PROPERTY ActualVelocity : REFERENCE TO LREAL
GET
ActualVelocity REF= lrActualVelocity;
END_GET
END_PROPERTY

PROPERTY AxisErrorID : REFERENCE TO UDINT
GET
AxisErrorID REF= iAxisErrorID;
END_GET
END_PROPERTY

PROPERTY AxisRef : AXIS_REF
GET
AxisRef := stAxisRef;
END_GET
SET
stAxisRef := AxisRef;
END_SET
END_PROPERTY

PROPERTY BufferMode : Tc2_MC2.MC_BufferMode
GET
BufferMode := eBufferMode;
END_GET
SET
eBufferMode := BufferMode;
END_SET
END_PROPERTY

PROPERTY Busy : REFERENCE TO BOOL
GET
Busy REF= bBusy;
END_GET
END_PROPERTY

PROPERTY Coupled : REFERENCE TO BOOL
GET
END_GET
END_PROPERTY

PROPERTY Deceleration : LREAL
GET
Deceleration := lrDeceleration;
END_GET
SET
lrDeceleration := Deceleration;
END_SET
END_PROPERTY

PROPERTY Direction : Tc2_MC2.MC_Direction
GET
Direction := eDirection;
END_GET
SET
eDirection := Direction;
END_SET
END_PROPERTY

PROPERTY Error : REFERENCE TO BOOL
GET
Error REF= bError;
END_GET
END_PROPERTY

PROPERTY ErrorID : REFERENCE TO UDINT
GET
ErrorID REF= iErrorID;
END_GET
END_PROPERTY

PROPERTY Halted : REFERENCE TO BOOL
GET
Halted REF= bHalted;
END_GET
END_PROPERTY

PROPERTY InPosition : REFERENCE TO BOOL
GET
InPosition REF= bInPostion;
END_GET
END_PROPERTY

PROPERTY InVelocity : REFERENCE TO BOOL
GET
InVelocity REF= bInVelocity;
END_GET
END_PROPERTY

PROPERTY IsHomed : REFERENCE TO BOOL
GET
IsHomed REF= bIsHomed;
END_GET
END_PROPERTY

PROPERTY Jerk : LREAL
GET
Jerk := lrJerk;
END_GET
SET
lrJerk := Jerk;
END_SET
END_PROPERTY

PROPERTY JogAcceleration : LREAL
GET
JogAcceleration := lrJogAcceleration;
END_GET
SET
lrJogAcceleration := JogAcceleration;
END_SET
END_PROPERTY

PROPERTY JogDeceleration : LREAL
GET
JogDeceleration := lrJogDeceleration;
END_GET
SET
lrJogDeceleration := JogDeceleration;
END_SET
END_PROPERTY

PROPERTY JogDirection : E_AxisJogDirection
GET
JogDirection := eJogDirection;
END_GET
SET
eJogDirection := JogDirection;
END_SET
END_PROPERTY

PROPERTY JogDone : REFERENCE TO BOOL
GET
JogDone REF= bJogDone;
END_GET
END_PROPERTY

PROPERTY JogJerk : LREAL
GET
JogJerk := lrJogJerk;
END_GET
SET
lrJogJerk := JogJerk;
END_SET
END_PROPERTY

PROPERTY JogMode : Tc2_MC2.E_JogMode
GET
JogMode := eJogMode;
END_GET
SET
eJogMode := JogMode;
END_SET
END_PROPERTY

PROPERTY JogPosition : LREAL
GET
JogPosition := lrJogPosition;
END_GET
SET
lrJogPosition := JogPosition;
END_SET
END_PROPERTY

PROPERTY JogVelocity : LREAL
GET
JogVelocity := lrJogVelocity;
END_GET
SET
lrJogVelocity := JogVelocity;
END_SET
END_PROPERTY

PROPERTY LagError : LREAL
GET
LagError := stAxisRef.NcToPlc.PosDiff;
END_GET
END_PROPERTY

PROPERTY Locked : REFERENCE TO BOOL
GET
Locked REF= bLocked;
END_GET
END_PROPERTY

PROPERTY MoveActive : REFERENCE TO BOOL
GET
MoveActive REF= bMoveActive;
END_GET
END_PROPERTY

METHOD MR_Abort : BOOL
IF eAxisState >= AXIS_INITIALIZING THEN
	bAbort := TRUE;
	eAxisState := AXIS_ABORTING;
	fbMachineLogger.MR_AddLogs(CONCAT(sName,' : abort requested'));
	
ELSIF eAxisState = AXIS_UNINITIALIZED THEN
	bAbort 		:= FALSE;
	MR_Abort	:= TRUE;
	fbMachineLogger.MR_AddLogs(CONCAT(sName,' : abort done'));
	
END_IF
END_METHOD

METHOD MR_Couple : BOOL
VAR_INPUT
END_VAR
;
END_METHOD

METHOD MR_Decouple : BOOL
VAR_INPUT
END_VAR
;
END_METHOD

METHOD MR_FirstCycle
VAR_INPUT
	sName 				: STRING; 	(* Axis object name *)
	sMeasurementUnits	: STRING;	(* Measurement units used by axis *)
	bModulo				: BOOL;		(* Axis is periodic *)
END_VAR
THIS^.sName := sName;
THIS^.sUnit := sMeasurementUnits;
THIS^.bModulo := bModulo;
END_METHOD

METHOD MR_Halt : BOOL
IF eAxisState >= AXIS_IDLE AND eAxisState <> AXIS_HALT_DONE THEN
	IF NOT bHaltLog THEN 
		fbMachineLogger.MR_AddLogs(CONCAT(sName,' : halt requested'));
		bHaltLog := TRUE;
	END_IF
	
	bHalt := TRUE;
	eAxisState := AXIS_HALT;
	
ELSIF eAxisState = AXIS_HALT_DONE THEN
	bInPostion 	:= FALSE;
	bInVelocity := FALSE;
	bMoveActive := FALSE;
	bStopped 	:= FALSE;
	bHalted 	:= TRUE;
	bJogDone 	:= FALSE;
	
	bHalt		:= FALSE;
	MR_Halt 	:= TRUE;

	bHaltLog 	:= FALSE;
	fbMachineLogger.MR_AddLogs(CONCAT(sName,' : halt done'));
	
END_IF
END_METHOD

METHOD MR_Home : BOOL
VAR_INPUT
	lrHomePosition : LREAL;
END_VAR
IF eAxisState = AXIS_IDLE THEN
	THIS^.lrHomePosition := lrHomePosition;
	bIsHomed := FALSE;
	
	bHome := TRUE;
	eAxisState := AXIS_HOME;
	fbMachineLogger.MR_AddLogs(CONCAT(sName,' : home position requested'));
	
ELSIF eAxisState = AXIS_HOME_DONE THEN
	bIsHomed := TRUE;
	
	bHome := FALSE;
	MR_Home := TRUE;
	fbMachineLogger.MR_AddLogs(CONCAT(sName,' : home position done'));	
	
END_IF
END_METHOD

METHOD MR_Init : BOOL
IF eAxisState = AXIS_UNINITIALIZED THEN
	bInit := TRUE;
	fbMachineLogger.MR_AddLogs(CONCAT(sName,' : initialization requested'));
	
ELSIF eAxisState = AXIS_INITIALIZING AND eAxisStateInit = AXIS_INIT_DONE THEN
	//bPowerOn 	:= TRUE;
	bInPostion 	:= FALSE;
	bInVelocity := FALSE;
	bMoveActive := FALSE;
	bStopped 	:= FALSE;
	bHalted 	:= FALSE;
	bJogDone 	:= FALSE;

	bInit 		:= FALSE;
	MR_Init 	:= TRUE;
	
	fbMachineLogger.MR_AddLogs(CONCAT(sName,' : initialization done'));

END_IF
END_METHOD

METHOD MR_Jog : BOOL
VAR_INPUT
	bJogActive	  : BOOL;
END_VAR
THIS^.bJogActive := bJogActive;

IF eAxisState = AXIS_IDLE THEN
	bJog := TRUE;
	bInPostion 	:= FALSE;
	bInVelocity	:= FALSE;
	bMoveActive	:= TRUE;
	bStopped	:= FALSE;
	bHalted 	:= FALSE;
	bJogDone 	:= FALSE;
	
	eAxisState := AXIS_MOVE_JOG;
	fbMachineLogger.MR_AddLogs(CONCAT(sName,' : move jog requested'));	
	
ELSIF eAxisState = AXIS_MOVE_JOG_DONE THEN
	IF eJogMode = E_JogMode.MC_JOGMODE_INCHING OR eJogMode = E_JogMode.MC_JOGMODE_INCHING_MODULO THEN
		bInPostion 	:= TRUE;
	END_IF
	
	bInVelocity := FALSE;
	bMoveActive := FALSE;
	bStopped 	:= FALSE;
	bHalted 	:= FALSE;
	bJogDone 	:= TRUE;	

	bJog 		:= FALSE;
	MR_Jog 		:= TRUE;
	
	fbMachineLogger.MR_AddLogs(CONCAT(sName,' : move jog done'));		
	
END_IF
END_METHOD

METHOD MR_MoveAbsolute : BOOL
VAR_INPUT
	lrAbsolutePosition : LREAL;
END_VAR
IF eAxisState = AXIS_IDLE AND THIS^.lrActualPosition <> lrAbsolutePosition THEN
	THIS^.lrAbsolutePosition := lrAbsolutePosition;
	bMoveAbsolute := TRUE;
	bInPostion 	:= FALSE;
	bInVelocity := FALSE;
	bMoveActive := TRUE;
	bStopped 	:= FALSE;
	bHalted 	:= FALSE;
	bJogDone 	:= FALSE;
	
	eAxisState := AXIS_MOVE_ABSOLUTE;
	fbMachineLogger.MR_AddLogs(CONCAT(sName,' : move absolute requested'));		
	
ELSIF eAxisState = AXIS_MOVE_ABSOLUTE_DONE THEN
	bInPostion 		:= TRUE;
	bInVelocity		:= FALSE;
	bMoveActive 	:= FALSE;
	bStopped 		:= FALSE;
	bHalted			:= FALSE;
	bJogDone 		:= FALSE;
	
	bMoveAbsolute 	:= FALSE;
	MR_MoveAbsolute := TRUE;
	fbMachineLogger.MR_AddLogs(CONCAT(sName,' : move absolute done'));		
	
END_IF
END_METHOD

METHOD MR_MoveAdditive : BOOL
VAR_INPUT
	lrRelativeDistance : LREAL;
END_VAR
THIS^.lrRelativeDistance := lrRelativeDistance;
IF eAxisState = AXIS_IDLE AND THIS^.lrRelativeDistance <> 0.0 THEN
	bMoveAdditive := TRUE;
	bInPostion 	:= FALSE;
	bInVelocity := FALSE;
	bStopped 	:= FALSE;
	bHalted 	:= FALSE;
	bJogDone 	:= FALSE;
	
	bMoveActive := TRUE;
	eAxisState := AXIS_MOVE_ADDITIVE;
	fbMachineLogger.MR_AddLogs(CONCAT(sName,' : move additive requested'));		
	
ELSIF eAxisState = AXIS_MOVE_ADDITIVE_DONE THEN
	bInPostion 		:= TRUE;
	bInVelocity 	:= FALSE;
	bStopped 		:= FALSE;
	bHalted 		:= FALSE;
	bJogDone 		:= FALSE;
	
	bMoveAdditive 	:= FALSE;
	MR_MoveAdditive := TRUE;
	fbMachineLogger.MR_AddLogs(CONCAT(sName,' : move additive done'));		
	
END_IF
END_METHOD

METHOD MR_MoveRelative : BOOL
VAR_INPUT
	lrRelativeDistance : LREAL;
END_VAR
THIS^.lrRelativeDistance := lrRelativeDistance;
IF eAxisState = AXIS_IDLE AND THIS^.lrRelativeDistance <> 0.0 THEN
	bMoveRelative := TRUE;
	bInPostion 	:= FALSE;
	bInVelocity := FALSE;
	bMoveActive := TRUE;
	bStopped 	:= FALSE;
	bHalted 	:= FALSE;
	bJogDone 	:= FALSE;
	
	eAxisState := AXIS_MOVE_RELATIVE;
	fbMachineLogger.MR_AddLogs(CONCAT(sName,' : move relative requested'));			
	
ELSIF eAxisState = AXIS_MOVE_RELATIVE_DONE THEN
	bMoveRelative 	:= FALSE;
	MR_MoveRelative := TRUE;
	
	bInPostion 		:= TRUE;
	bInVelocity 	:= FALSE;
	bMoveActive 	:= FALSE;
	bStopped 		:= FALSE;
	bHalted 		:= FALSE;
	bJogDone 		:= FALSE;
	
	fbMachineLogger.MR_AddLogs(CONCAT(sName,' : move relative done'));		
	
END_IF
END_METHOD

METHOD MR_MoveVelocity : BOOL
IF eAxisState = AXIS_IDLE THEN
	bMoveVelocity 	:= TRUE;
	bInPostion 		:= FALSE;
	bInVelocity 	:= FALSE;
	bMoveActive 	:= TRUE;
	bStopped 		:= FALSE;
	bHalted 		:= FALSE;
	bJogDone 		:= FALSE;	
	
	eAxisState 		:= AXIS_MOVE_VELOCITY;
	fbMachineLogger.MR_AddLogs(CONCAT(sName,' : move velocity requested'));			
	
ELSIF eAxisState = AXIS_MOVE_VELOCITY_DONE THEN
	bMoveVelocity 	:= FALSE;
	MR_MoveVelocity := TRUE;
	
	bInPostion 		:= FALSE;
	bInVelocity 	:= TRUE;
	bMoveActive 	:= TRUE;
	bStopped 		:= FALSE;
	bHalted 		:= FALSE;
	bJogDone 		:= FALSE;
	
	fbMachineLogger.MR_AddLogs(CONCAT(sName,' : move velocity done'));		
	
END_IF
END_METHOD

METHOD MR_Reset : BOOL
IF eAxisState <> AXIS_RESET AND eAxisState <> AXIS_RESET_DONE AND bError THEN
	bReset := TRUE;
	eAxisStateBeforeReset := eAxisState;
	eAxisState := AXIS_RESET;
	fbMachineLogger.MR_AddLogs(CONCAT(sName,' : reset requested'));			
	
ELSIF eAxisState = AXIS_RESET_DONE THEN
	bError := FALSE;
	iErrorID := 0;
	
	bReset := FALSE;
	MR_Reset := TRUE;
	
	fbMachineLogger.MR_AddLogs(CONCAT(sName,' : reset done'));		
		
END_IF
END_METHOD

METHOD MR_Stop : BOOL
IF eAxisState >= AXIS_IDLE AND eAxisState <> AXIS_STOP_DONE THEN
	IF NOT bStopLog THEN 
		fbMachineLogger.MR_AddLogs(CONCAT(sName,' : stop requested'));
		bStopLog := TRUE;	
	END_IF
	
	bStop := TRUE;
	eAxisState := AXIS_STOP;
	
ELSIF eAxisState = AXIS_STOP_DONE THEN
	bStop 		:= FALSE;
	MR_Stop 	:= TRUE;
	
	bInPostion 	:= FALSE;
	bInVelocity := FALSE;
	bMoveActive := FALSE;
	bStopped 	:= TRUE;
	bHalted 	:= FALSE;
	bJogDone 	:= FALSE;
	bLocked		:= TRUE;
	
	bStopLog 	:= FALSE;
	fbMachineLogger.MR_AddLogs(CONCAT(sName,' : stop done'));			
END_IF
END_METHOD

METHOD MR_Unlock : BOOL
VAR_INPUT
END_VAR
IF eAxisState = AXIS_IDLE THEN
	bUnlock := TRUE;
	MR_Unlock := FALSE;
	eAxisState := AXIS_UNLOCK;
	fbMachineLogger.MR_AddLogs(CONCAT(sName,' : unlock after stop requested'));
	
ELSIF eAxisState = AXIS_UNLOCK_DONE THEN
	bUnlock := FALSE;
	MR_Unlock := TRUE;
	bLocked := FALSE;
	fbMachineLogger.MR_AddLogs(CONCAT(sName,' : unlock after stop done'));
	
END_IF
END_METHOD

METHOD PROTECTED MS_Aborting
VAR_INPUT
END_VAR
(* Reset MC_Halt *)
fbMcHalt( Axis := stAxisRef, Execute := FALSE);

(* Reset MC_Stop *)
fbMcStop( Axis := stAxisRef, Execute := FALSE);

(* Reset MC_MoveVelocity *)
fbMcMoveVelocity( Axis := stAxisRef, Execute := FALSE);

(* Reset MC_MoveAbsolute *)
fbMcMoveAbsolute( Axis := stAxisRef, Execute := FALSE);

(* Reset MC_MoveAdditive *)
fbMcMoveAdditive( Axis := stAxisRef, Execute := FALSE);

(* Reset MC_MoveRelative *)
fbMcMoveRelative( Axis := stAxisRef, Execute := FALSE);

(* Reset MC_Jog *)
fbMcJog( Axis := stAxisRef, JogForward := FALSE ,JogBackwards := FALSE);

(* Reset MC_Reset *)
fbMcReset( Axis := stAxisRef, Execute := FALSE);

(* Reset MC_Power *)
fbMcPower(	Enable 			:= FALSE,
			Enable_Positive := FALSE,
			Enable_Negative := FALSE,
			Override 		:= lrOverride,
			Axis 			:= stAxisRef);
					
IF fbReadAxisStatus.Disabled AND NOT fbMcStop.Busy THEN
	bInPostion	:= FALSE;
	bInVelocity := FALSE;
	bMoveActive := FALSE;
	bStopped 	:= FALSE;
	bHalted 	:= FALSE;
	bJogDone	:= FALSE;
	bIsHomed 	:= FALSE;
	bLocked		:= FALSE;
	eAxisState	:= AXIS_UNINITIALIZED;	
	
END_IF
END_METHOD

METHOD PROTECTED MS_Couple : BOOL
VAR_INPUT
END_VAR
(*
IF NOT fbMcGearIn.Error THEN
	fbMcGearIn( Master				:=,
				Slave 				:= ,
				Execute 			:= TRUE,
				RatioNumerator		:=,
				RatioDenominator 	:=,
				Acceleration 		:= ,
				Deceleration 		:= ,
				Jerk 				:=,
				BufferMode 			:=,
				Options				:=);
				
	IF fbMcGearIn.InGear THEN
		eAxisState := AXIS_COUPLE_DONE;
	END_IF
ELSE
	bError := TRUE;
	iErrorID := fbMcGearIn.ErrorID;
	fbMcGearIn( Master := , Slave := , Execute := FALSE);
	fbAlarmCoupling.ipArguments.Clear().AddUDInt(iErrorID);
	fbAlarmCoupling.Raise(0);
END_IF
*)
END_METHOD

METHOD MS_CoupleDone : BOOL
VAR_INPUT
END_VAR
END_METHOD

METHOD MS_Decouple : BOOL
VAR_INPUT
END_VAR
(*
IF NOT fbMcGearOut.Error THEN			
	fbMcGearOut( 	Slave 	:=,
					Execute := TRUE,
					Options := );	
				
	IF fbMcGearOut.Done THEN
		eAxisState := AXIS_DECOUPLE_DONE;
	END_IF
ELSE
	bError := TRUE;
	iErrorID := fbMcGearOut.ErrorID;
	fbMcGearOut( Slave := , Execute := FALSE);
	fbAlarmDecoupling.ipArguments.Clear().AddUDInt(iErrorID);
	fbAlarmDecoupling.Raise(0);
END_IF
*)
END_METHOD

METHOD MS_DecoupleDone : BOOL
VAR_INPUT
END_VAR
END_METHOD

METHOD MS_Extension : BOOL
VAR_INPUT
END_VAR
END_METHOD

METHOD PROTECTED MS_Halt
VAR_INPUT
END_VAR
(* Reset MC_MoveVelocity *)
fbMcMoveVelocity( Axis := stAxisRef, Execute := FALSE);

(* Reset MC_MoveAbsolute *)					
fbMcMoveAbsolute( Axis := stAxisRef, Execute := FALSE);

(* Reset MC_MoveAdditive *)					
fbMcMoveAdditive( Axis := stAxisRef ,Execute := FALSE);

(* Reset MC_MoveRelative *)					
fbMcMoveRelative( Axis := stAxisRef, Execute := FALSE);

(* Reset MC_Jog *)
fbMcJog( Axis := stAxisRef, JogForward := FALSE, JogBackwards := FALSE);

fbMcHalt(	Axis			:= stAxisRef,
			Execute 		:= TRUE,
			Deceleration 	:= lrDeceleration,
			Jerk 			:= lrJerk,
			BufferMode 		:= MC_Aborting);

IF fbMcHalt.Error THEN
	bError := TRUE;
	iErrorID := fbMcHalt.ErrorID;
	fbMcHalt(Axis := stAxisRef, Execute := FALSE);
	fbAlarmHalt.ipArguments.Clear().AddUDInt(iErrorID);
	fbAlarmHalt.Raise(0);

ELSIF fbMcHalt.Done THEN
	eAxisState := AXIS_HALT_DONE;
END_IF
END_METHOD

METHOD PROTECTED MS_HaltDone
VAR_INPUT
END_VAR
fbMcHalt( Axis := stAxisRef, Execute := FALSE);

IF NOT bHalt AND NOT fbMcHalt.Busy THEN
	eAxisState := AXIS_IDLE;
END_IF
END_METHOD

METHOD PROTECTED ABSTRACT MS_Home
VAR_INPUT
END_VAR
END_METHOD

METHOD PROTECTED ABSTRACT MS_HomeDone
VAR_INPUT
END_VAR
END_METHOD

METHOD PROTECTED MS_Idle
VAR_INPUT
END_VAR
;
END_METHOD

METHOD PROTECTED MS_Initializing
VAR_INPUT
END_VAR
CASE eAxisStateInit OF
	AXIS_INIT_RESET:
		fbMcReset(	Execute := TRUE, Axis := stAxisRef);
		
		IF fbMcReset.Error THEN
			bError := fbMcReset.Error;
			iErrorID := fbMcReset.ErrorID;
			fbMcReset(Axis := stAxisRef, Execute := FALSE);
			fbAlarmInitReset.ipArguments.Clear().AddUDInt(iErrorID);
			fbAlarmInitReset.Raise(0);
			
		ELSIF fbMcReset.Done THEN
			fbMcReset(Axis := stAxisRef, Execute := FALSE);
			eAxisStateInit := AXIS_INIT_POWER_ON;
			
		END_IF
		
	AXIS_INIT_POWER_ON:
		fbMcPower(	Enable 			:= TRUE,
					Enable_Positive := TRUE,
					Enable_Negative := TRUE,
					Override 		:= lrOverride,
					Axis 			:= stAxisRef);
			
		IF fbMcPower.Error THEN
			bError := fbMcPower.Error;
			iErrorID := fbMcPower.ErrorID;
			fbAlarmInitPowerOn.ipArguments.Clear().AddUDInt(iErrorID);
			fbAlarmInitPowerOn.Raise(0);			
			
		ELSIF fbMcPower.Status THEN
			eAxisStateInit := AXIS_INIT_DONE;	
				
		END_IF
	
	AXIS_INIT_DONE:
		IF NOT bInit THEN
			eAxisState := AXIS_READY_INITIALIZED;
		END_IF
END_CASE
END_METHOD

METHOD PROTECTED MS_MoveAbsolute
VAR_INPUT
END_VAR
fbMcMoveAbsolute(	Axis			:= stAxisRef,
					Execute 		:= TRUE,
					Position 		:= lrAbsolutePosition,
					Velocity 		:= lrVelocity,
					Acceleration 	:= lrAcceleration,
					Deceleration 	:= lrDeceleration,
					Jerk 			:= lrJerk,
					BufferMode 		:= eBufferMode);

IF fbMcMoveAbsolute.Error THEN
	bError := TRUE;
	bMoveActive := FALSE;
	iErrorID := fbMcMoveAbsolute.ErrorID;
	fbMcMoveAbsolute( Axis := stAxisRef, Execute := FALSE);
	fbAlarmMoveAbsolute.ipArguments.Clear().AddUDInt(iErrorID);
	fbAlarmMoveAbsolute.Raise(0);

ELSIF fbMcMoveAbsolute.Done THEN
	eAxisState := AXIS_MOVE_ABSOLUTE_DONE;
END_IF
END_METHOD

METHOD PROTECTED MS_MoveAbsoluteDone
VAR_INPUT
END_VAR
fbMcMoveAbsolute( Axis := stAxisRef, Execute := FALSE);

IF NOT bMoveAbsolute AND NOT fbMcMoveAbsolute.Busy THEN
	eAxisState := AXIS_IDLE;
END_IF
END_METHOD

METHOD PROTECTED MS_MoveAdditive
VAR_INPUT
END_VAR
fbMcMoveAdditive(	Axis			:= stAxisRef,
					Execute 		:= TRUE,
					Distance 		:= lrRelativeDistance,
					Velocity		:= lrVelocity,
					Acceleration	:= lrAcceleration,
					Deceleration	:= lrDeceleration,
					Jerk			:= lrJerk,
					BufferMode 		:= eBufferMode);

IF fbMcMoveAdditive.Error THEN
	bError := TRUE;
	bMoveActive := FALSE;
	iErrorID := fbMcMoveAdditive.ErrorID;
	fbMcMoveAdditive( Axis := stAxisRef, Execute := FALSE);
	fbAlarmMoveAdditive.ipArguments.Clear().AddUDInt(iErrorID);
	fbAlarmMoveAdditive.Raise(0);
		
ELSIF fbMcMoveAdditive.Done THEN
	eAxisState := AXIS_MOVE_ADDITIVE_DONE;
END_IF
END_METHOD

METHOD PROTECTED MS_MoveAdditiveDone
VAR_INPUT
END_VAR
fbMcMoveAdditive( Axis := stAxisRef, Execute := FALSE);

IF NOT bMoveAdditive AND NOT fbMcMoveAdditive.Busy THEN
	eAxisState := AXIS_IDLE;
END_IF
END_METHOD

METHOD PROTECTED MS_MoveJog
VAR_INPUT
END_VAR
VAR
	bJogForward: BOOL;
	bJogBackward: BOOL;
END_VAR
IF eJogDirection = AXIS_JOG_DIR_POSITIVE THEN
	bJogForward := TRUE;
	bJogBackward:= FALSE;
	
ELSIF eJogDirection = AXIS_JOG_DIR_NEGATIVE THEN
	bJogForward := FALSE;
	bJogBackward:= TRUE;
		
END_IF

fbMcJog( 	Axis 			:= stAxisRef,
			JogForward		:= bJogForward,
			JogBackwards	:= bJogBackward,
			Mode 			:= eJogMode,
			Position 		:= lrJogPosition,
			Velocity 		:= lrJogVelocity,
			Acceleration 	:= lrJogAcceleration,
			Deceleration 	:= lrJogDeceleration,
			Jerk 			:= lrJogJerk);

IF fbMcJog.Error THEN
	bError := TRUE;
	bMoveActive := FALSE;
	iErrorID := fbMcJog.ErrorID;
	fbMcJog( Axis := stAxisRef, JogForward := FALSE, JogBackwards := FALSE);
	fbAlarmMoveJog.ipArguments.Clear().AddUDInt(iErrorID);
	fbAlarmMoveJog.Raise(0);
	
ELSIF fbMcJog.Mode >= MC_JOGMODE_INCHING AND fbMcJog.Done THEN
	eAxisState := AXIS_MOVE_JOG_DONE;
		
ELSIF fbMcJog.Mode < MC_JOGMODE_INCHING AND NOT bJogActive THEN
	eAxisState := AXIS_MOVE_JOG_DONE;
		
END_IF
END_METHOD

METHOD PROTECTED MS_MoveJogDone
VAR_INPUT
END_VAR
fbMcJog( Axis := stAxisRef, JogForward := FALSE, JogBackwards := FALSE);

IF NOT bJog AND NOT fbMcJog.Busy THEN
	eAxisState := AXIS_IDLE;
END_IF
END_METHOD

METHOD PROTECTED MS_MoveRelative
VAR_INPUT
END_VAR
fbMcMoveRelative(	Axis 			:= stAxisRef,
					Execute 		:= TRUE,
					Distance 		:= lrRelativeDistance,
					Velocity 		:= lrVelocity,
					Acceleration 	:= lrAcceleration,
					Deceleration 	:= lrDeceleration,
					Jerk 			:= lrJerk,
					BufferMode 		:= eBufferMode);
				
IF fbMcMoveRelative.Error THEN
	bError := TRUE;
	iErrorID := fbMcMoveRelative.ErrorID;
	fbMcMoveRelative( Axis := stAxisRef, Execute := FALSE);
	fbAlarmMoveRelative.ipArguments.Clear().AddUDInt(iErrorID);
	fbAlarmMoveRelative.Raise(0);
	
ELSIF fbMcMoveRelative.Done THEN
	eAxisState := AXIS_MOVE_RELATIVE_DONE;
END_IF
END_METHOD

METHOD PROTECTED MS_MoveRelativeDone
VAR_INPUT
END_VAR
fbMcMoveRelative( Axis := stAxisRef, Execute := FALSE);

IF NOT bMoveRelative AND NOT fbMcMoveRelative.Busy THEN
	bInPostion := TRUE;
	bInVelocity := FALSE;
	bMoveActive := FALSE;
	bStopped := FALSE;
	bHalted := FALSE;
	bJogDone := FALSE;
	eAxisState := AXIS_IDLE;
END_IF
END_METHOD

METHOD PROTECTED MS_MoveVelocity
VAR_INPUT
END_VAR
fbMcMoveVelocity(	Axis 			:= stAxisRef,
					Execute 		:= TRUE,
					Velocity 		:= lrVelocity,
					Acceleration 	:= lrAcceleration,
					Deceleration 	:= lrDeceleration,
					Jerk 			:= lrJerk,
					Direction 		:= eDirection,
					BufferMode 		:= eBufferMode);

IF fbMcMoveVelocity.Error THEN
	bError := TRUE;
	iErrorID := fbMcMoveVelocity.ErrorID;
	fbMcMoveVelocity( Axis := stAxisRef, Execute := FALSE);
	fbAlarmMoveVelocity.ipArguments.Clear().AddUDInt(iErrorID);
	fbAlarmMoveVelocity.Raise(0);
	
ELSIF fbMcMoveVelocity.InVelocity THEN
	eAxisState := AXIS_MOVE_VELOCITY_DONE;
END_IF
END_METHOD

METHOD PROTECTED MS_MoveVelocityDone
VAR_INPUT
END_VAR
fbMcMoveVelocity( Axis := stAxisRef, Execute := FALSE);

IF NOT bMoveVelocity AND NOT fbMcMoveVelocity.Busy THEN
	eAxisState := AXIS_IDLE;
END_IF
END_METHOD

METHOD PROTECTED MS_ReadyInitialized
VAR_INPUT
END_VAR
eAxisState := AXIS_IDLE;
END_METHOD

METHOD PROTECTED MS_Reset
VAR_INPUT
END_VAR
(* Reset MC_Halt *)
fbMcHalt( Axis := stAxisRef, Execute := FALSE);

(* Reset MC_Stop *)
fbMcStop( Axis := stAxisRef, Execute := FALSE);

(* Reset MC_MoveVelocity *)
fbMcMoveVelocity( Axis := stAxisRef, Execute := FALSE);

(* Reset MC_MoveAbsolute *)
fbMcMoveAbsolute( Axis := stAxisRef, Execute := FALSE);

(* Reset MC_MoveAdditive *)
fbMcMoveAdditive( Axis := stAxisRef, Execute := FALSE);

(* Reset MC_MoveRelative *)
fbMcMoveRelative( Axis := stAxisRef, Execute := FALSE);

(* Reset MC_Jog *)
fbMcJog( Axis := stAxisRef, JogForward := FALSE ,JogBackwards := FALSE);

(* Reset MC_GearIn *)
;

(* Reset MC_GearOut *)
;

(* Reset internal commands *)
bAbort			:= FALSE;
bHalt 			:= FALSE;
bHome			:= FALSE;
bJog			:= FALSE;
bMoveAbsolute	:= FALSE;
bMoveAdditive	:= FALSE;
bMoveRelative	:= FALSE;
bMoveVelocity	:= FALSE;
bStop			:= FALSE;

fbMcReset( Axis := stAxisRef, Execute := TRUE);

IF fbMcReset.Error THEN
	bError := TRUE;
	iErrorID := fbMcReset.ErrorID;
	fbMcReset( Axis := stAxisRef, Execute := FALSE);
	fbAlarmInitReset.ipArguments.Clear().AddUDInt(iErrorID);
	fbAlarmInitReset.Raise(0);
	
ELSIF fbMcReset.Done THEN
	fbMcReset(Axis := stAxisRef, Execute := FALSE);
	
	(* Confirming and resetting alarms *)
	fbAlarmHalt.Confirm(nTimeStamp := 0);
	fbAlarmInitReset.Confirm(nTimeStamp := 0);
	fbAlarmInitPowerOn.Confirm(nTimeStamp := 0);
	fbAlarmMoveAbsolute.Confirm(nTimeStamp := 0);
	fbAlarmMoveAdditive.Confirm(nTimeStamp := 0);
	fbAlarmMoveJog.Confirm(nTimeStamp := 0);
	fbAlarmMoveRelative.Confirm(nTimeStamp := 0);
	fbAlarmMoveVelocity.Confirm(nTimeStamp := 0);
	fbAlarmStop.Confirm(nTimeStamp := 0);
	fbAlarmHome.Confirm(nTimeStamp := 0);
	fbAlarmHaltCA.Confirm(nTimeStamp := 0);
	fbAlarmMoveAbsoluteCA.Confirm(nTimeStamp := 0);
	fbAlarmMoveRelativeCA.Confirm(nTimeStamp := 0);
	fbAlarmCoupling.Confirm(nTimeStamp := 0);
	fbAlarmDecoupling.Confirm(nTimeStamp := 0);

	fbAlarmHalt.Clear(nTimeStamp := 0, bResetConfirmation := bResetConfirmation); 
	fbAlarmInitReset.Clear(nTimeStamp := 0, bResetConfirmation := bResetConfirmation); 
	fbAlarmInitPowerOn.Clear(nTimeStamp := 0, bResetConfirmation := bResetConfirmation); 
	fbAlarmMoveAbsolute.Clear(nTimeStamp := 0, bResetConfirmation := bResetConfirmation); 
	fbAlarmMoveAdditive.Clear(nTimeStamp := 0, bResetConfirmation := bResetConfirmation); 
	fbAlarmMoveJog.Clear(nTimeStamp := 0, bResetConfirmation := bResetConfirmation); 
	fbAlarmMoveRelative.Clear(nTimeStamp := 0, bResetConfirmation := bResetConfirmation); 
	fbAlarmMoveVelocity.Clear( nTimeStamp := 0, bResetConfirmation := bResetConfirmation); 
	fbAlarmStop.Clear(nTimeStamp := 0, bResetConfirmation := bResetConfirmation); 
	fbAlarmHome.Clear(nTimeStamp := 0, bResetConfirmation := bResetConfirmation); 
	fbAlarmHaltCA.Clear(nTimeStamp := 0, bResetConfirmation := bResetConfirmation); 
	fbAlarmMoveAbsoluteCA.Clear(nTimeStamp := 0, bResetConfirmation := bResetConfirmation); 
	fbAlarmMoveRelativeCA.Clear(nTimeStamp := 0, bResetConfirmation := bResetConfirmation); 
	fbAlarmCoupling.Clear(nTimeStamp := 0, bResetConfirmation := bResetConfirmation); 
	fbAlarmDecoupling.Clear(nTimeStamp := 0, bResetConfirmation := bResetConfirmation); 

	IF NOT fbMcHalt.Busy AND NOT fbMcStop.Busy AND NOT fbMcMoveVelocity.Busy AND
		NOT fbMcMoveAbsolute.Busy AND NOT fbMcMoveAdditive.Busy AND NOT fbMcMoveRelative.Busy AND NOT fbMcReset.Busy THEN
		eAxisState := AXIS_RESET_DONE;
	END_IF
END_IF
END_METHOD

METHOD PROTECTED MS_ResetDone
VAR_INPUT
END_VAR
IF NOT bReset THEN
	IF eAxisStateBeforeReset >= E_AxisState.AXIS_IDLE THEN
		eAxisState := AXIS_IDLE;
	ELSE
		eAxisState := AXIS_UNINITIALIZED;	
	END_IF
END_IF
END_METHOD

METHOD PROTECTED MS_Stop
VAR_INPUT
END_VAR
(* Reset MC_MoveVelocity *)
fbMcMoveVelocity( Axis := stAxisRef, Execute := FALSE);

(* Reset MC_MoveAbsolute *)					
fbMcMoveAbsolute( Axis := stAxisRef, Execute := FALSE);

(* Reset MC_MoveAdditive *)					
fbMcMoveAdditive( Axis := stAxisRef ,Execute := FALSE);

(* Reset MC_MoveRelative *)					
fbMcMoveRelative( Axis := stAxisRef, Execute := FALSE);

(* Reset MC_Jog *)
fbMcJog( Axis := stAxisRef, JogForward := FALSE, JogBackwards := FALSE);

fbMcStop(	Execute 		:= TRUE,
			Axis 			:= stAxisRef,
			Deceleration	:= lrStopDeceleration,
			Jerk 			:= lrStopJerk);

IF fbMcStop.Error THEN
	bError := TRUE;
	iErrorID := fbMcStop.ErrorID;
	fbMcStop( Axis := stAxisRef, Execute := FALSE);
	fbAlarmStop.ipArguments.Clear().AddUDInt(iErrorID);
	fbAlarmStop.Raise(0);
	
ELSIF fbMcStop.Done THEN
	eAxisState := AXIS_STOP_DONE;
END_IF
END_METHOD

METHOD PROTECTED MS_StopDone
VAR_INPUT
END_VAR
fbMcStop( Axis := stAxisRef, Execute := FALSE);

IF NOT bStop THEN
	eAxisState := AXIS_IDLE;	
END_IF
END_METHOD

METHOD PROTECTED MS_Uninitalized
VAR_INPUT
END_VAR
(* Reset all commands *)
bAbort				:= FALSE;
bHalt 				:= FALSE;
bHome				:= FALSE;
bJog				:= FALSE;
bMoveAbsolute		:= FALSE;
bMoveAdditive		:= FALSE;
bMoveRelative		:= FALSE;
bMoveVelocity		:= FALSE;
bReset				:= FALSE;
bStop				:= FALSE;

(* Reset status flags *)
bError				:= FALSE;
bInPostion			:= FALSE;
bInVelocity			:= FALSE;
bIsHomed			:= FALSE;
bMoveActive			:= FALSE;
bPowerOn			:= FALSE;
bStopped			:= FALSE;
bJogDone			:= FALSE;
bLocked				:= FALSE;
lrActualPosition 	:= 0.0;
lrActualVelocity 	:= 0.0;
iErrorID			:= 0;

IF bInit THEN
	eAxisState := AXIS_INITIALIZING;
	eAxisStateInit := AXIS_INIT_RESET;	
END_IF
END_METHOD

METHOD MS_Unlock
VAR_INPUT
END_VAR
fbMcStop( Axis := stAxisRef, Execute := FALSE);

IF NOT fbMcStop.Busy THEN
	eAxisState := AXIS_UNLOCK_DONE;
END_IF
END_METHOD

METHOD MS_UnlockDone
VAR_INPUT
END_VAR
IF NOT bUnlock THEN
	eAxisState := AXIS_IDLE;
END_IF
END_METHOD

PROPERTY Name : STRING
GET
Name := sName;
END_GET
SET
sName := Name;
END_SET
END_PROPERTY

PROPERTY Options : Tc2_MC2.ST_MoveOptions
GET
Options := stOptions;
END_GET
SET
stOptions := Options;
END_SET
END_PROPERTY

PROPERTY Override : LREAL
GET
Override := lrOverride;
END_GET
SET
IF Override >= 0.0 AND Override <= 200.0 THEN
	lrOverride := Override;
	fbMcPower( Axis := stAxisRef, Override := lrOverride);
END_IF
END_SET
END_PROPERTY

PROPERTY PowerOn : REFERENCE TO BOOL
GET
PowerOn REF= bPowerOn;
END_GET
END_PROPERTY

PROPERTY SetpointPosition : LREAL
GET
SetpointPosition := stAxisRef.NcToPlc.SetPos;
END_GET
END_PROPERTY

PROPERTY SetpointVelocity : LREAL
GET
SetpointVelocity := stAxisRef.NcToPlc.SetVelo;
END_GET
END_PROPERTY

PROPERTY State : REFERENCE TO E_AxisState
GET
State REF= eAxisState;
END_GET
END_PROPERTY

METHOD PROTECTED StateMachine
VAR_INPUT
END_VAR

VAR

END_VAR
CASE eAxisState OF
	AXIS_UNINITIALIZED:
		MS_Uninitalized();
		
	AXIS_INITIALIZING:
		MS_Initializing();
		
	AXIS_READY_INITIALIZED:
		MS_ReadyInitialized();
		
	AXIS_IDLE:
		MS_Idle();
	
	AXIS_HOME:
		MS_Home();
		
	E_AxisState.AXIS_HOME_DONE:
		MS_HomeDone();
		
	AXIS_MOVE_VELOCITY:
		MS_MoveVelocity();
	
	AXIS_MOVE_VELOCITY_DONE:
		MS_MoveVelocityDone();
	
	AXIS_MOVE_ABSOLUTE:
		MS_MoveAbsolute();
	
	AXIS_MOVE_ABSOLUTE_DONE:
		MS_MoveAbsoluteDone();
	
	AXIS_MOVE_ADDITIVE:
		MS_MoveAdditive();
	
	AXIS_MOVE_ADDITIVE_DONE:
		MS_MoveAdditiveDone();
		
	AXIS_MOVE_RELATIVE:
		MS_MoveRelative();
		
	AXIS_MOVE_RELATIVE_DONE:
		MS_MoveRelativeDone();
	
	AXIS_MOVE_JOG:
		MS_MoveJog();
	
	AXIS_MOVE_JOG_DONE:
		MS_MoveJogDone();
	
	AXIS_STOP:
		MS_Stop();
	
	AXIS_STOP_DONE:
		MS_StopDone();
		
	AXIS_HALT:
		MS_Halt();
	
	AXIS_HALT_DONE:
		MS_HaltDone();	
	
	AXIS_RESET:
		MS_Reset();
	
	AXIS_RESET_DONE:
		MS_ResetDone();
		
	AXIS_ABORTING:
		MS_Aborting();
		
	AXIS_COUPLE:
		MS_Couple();
		
	AXIS_COUPLE_DONE:
		MS_CoupleDone();
		
	AXIS_DECOUPLE:
		MS_Decouple();
		
	AXIS_DECOUPLE_DONE:
		MS_DecoupleDone();
		
	AXIS_UNLOCK:
		MS_Unlock();
	
	AXIS_UNLOCK_DONE:
		MS_UnlockDone();
		
	AXIS_EXTENSION:
		MS_Extension();
		
END_CASE
END_METHOD

PROPERTY StatePlcOpen : REFERENCE TO E_AxisStatePlcOpen
GET
StatePlcOpen REF= eStatePlcOpen;
END_GET
END_PROPERTY

PROPERTY StopDeceleration : LREAL
GET
StopDeceleration := lrStopDeceleration;
END_GET
SET
lrStopDeceleration := StopDeceleration;
END_SET
END_PROPERTY

PROPERTY StopJerk : LREAL
GET
StopJerk := lrStopJerk;
END_GET
SET
lrStopJerk := StopJerk;
END_SET
END_PROPERTY

PROPERTY Stopped : REFERENCE TO BOOL
GET
Stopped REF= bStopped;
END_GET
END_PROPERTY

PROPERTY Unit : STRING
GET
Unit := sUnit;
END_GET
SET
sUnit := Unit;
END_SET
END_PROPERTY

PROPERTY Velocity : LREAL
GET
Velocity := lrVelocity;
END_GET
SET
lrVelocity := Velocity;
END_SET
END_PROPERTY

END_FUNCTION_BLOCK

// ---- POUs/Libs/Digital Devices/Digital Input/FB_DigitalInput.TcPOU
(* 
| :Description: This function block represents basic digital input and can be used for creating an instance of signle digital input device like buttons, switches, sensors.
| To get the current status of digital input use "Value" property. To simulate state of the input by software set "Enable Force" parameter and change value via "MR_ResetForceValue" and "MR_SetForceValue" methods.
*)
FUNCTION_BLOCK FB_DigitalInput EXTENDS FB_DigitalDevice IMPLEMENTS I_DigitalInput
VAR
	(* Internal status *)
	bIn				AT %I*	: BOOL;		(* Current value of input *)
	bInForced				: BOOL;		(* Forced value from software *)
	bEnableForce			: BOOL;		(* Enable forcing of the input from software *)
	bRisingTrigger 			: BOOL;		(* Rising trigger of input detected*)
	bFallingTrigger 		: BOOL;		(* Falling trigger of input detected*)
	
	(* Function blocks *)
	rtRisingTrigger 		: R_TRIG;	(* Rising trigger detecting FB*)
	ftFallingTrigger		: F_TRIG;	(* Falling trigger detecting FB*)
END_VAR
(*
Version history:

+-------------+------------+----------------+----------+------------------------------------------+
|Date         | Version    | created under  | Author   | Remark                                   |
+=============+============+================+==========+==========================================+
|2021-11      | 1.0.0.0    | V3.1.4024.22   | ADBO     | Function block created                   |
+-------------+------------+----------------+----------+------------------------------------------+
|2022-01      | 1.1.0.0    | V3.1.4024.22   | ADBO     | Changed to child of FB_DigitalDevice     |
+-------------+------------+----------------+----------+------------------------------------------+

*)

PROPERTY EnableForce : BOOL
GET
EnableForce := bEnableForce;
END_GET
SET
bEnableForce := EnableForce;
END_SET
END_PROPERTY

PROPERTY FallingTrigger : BOOL
GET
ftFallingTrigger(CLK := In, Q => bFallingTrigger);
FallingTrigger := bFallingTrigger;
END_GET
END_PROPERTY

PROPERTY In : BOOL
GET
IF NOT bEnableForce THEN
	In := bIn;
ELSE
	In := bInForced;
END_IF
END_GET
END_PROPERTY

METHOD MR_ResetForceValue
IF bEnableForce THEN
	bInForced := FALSE;
	
END_IF
END_METHOD

METHOD MR_SetForceValue
IF bEnableForce THEN
	bInForced := TRUE;
	
END_IF
END_METHOD

PROPERTY RisingTrigger : BOOL
GET
rtRisingTrigger(CLK := In, Q => bRisingTrigger);
RisingTrigger := bRisingTrigger;
END_GET
END_PROPERTY

END_FUNCTION_BLOCK

// ---- POUs/Libs/Digital Devices/Digital Device/FB_DigitalDevice.TcPOU
(* 
:Description: This function block is base for all other digital devices.
*)
FUNCTION_BLOCK ABSTRACT FB_DigitalDevice IMPLEMENTS I_DigitalDevice
VAR
	sName : STRING; (* Name of digital device instance *)
	sModuleType : STRING;
	sPortID		: STRING;
END_VAR
(*
Version history:

+-------------+------------+----------------+----------+------------------------------------------+
|Date         | Version    | created under  | Author   | Remark                                   |
+=============+============+================+==========+==========================================+
|2022-01      | 1.0.0.0    | V3.1.4024.22   | ADBO     | Function block created                   |
+-------------+------------+----------------+----------+------------------------------------------+

*)

PROPERTY ModuleType : REFERENCE TO STRING
GET
ModuleType REF= sModuleType;
END_GET
END_PROPERTY

METHOD MR_FirstCycle : BOOL
VAR_INPUT
	sName : STRING;
	sModuleType : STRING;
	sPortID		: STRING;
END_VAR
THIS^.sName := sName;
THIS^.sModuleType := sModuleType;
THIS^.sPortID := sPortID;
END_METHOD

PROPERTY Name : REFERENCE TO STRING
GET
Name REF= sName;
END_GET
END_PROPERTY

PROPERTY PortID : REFERENCE TO STRING
GET
PortID REF= sPortID;
END_GET
END_PROPERTY

END_FUNCTION_BLOCK

// ---- POUs/Libs/Communication/TcpIp/FUN_StringToTcpBufferData.TcPOU
(* :Description:  This function is used to convert string into bytes structure, ready to send it via TCP/IP protocole *)
FUNCTION FUN_StringToTcpBufferData : BOOL
VAR_INPUT
	sMessageAddr 	: PVOID;					(* Source string message *)
	stSendDataAddr	: PVOID;					(* Destination TCP/IP data structure *)
END_VAR
VAR
	psMessage	: POINTER TO STRING;			(* Pointer to string converted to structure *)
	pstSendData	: POINTER TO ST_TcpBufferData;	(* Pointer to structure made of string bytes *)
END_VAR
(*
Version history:

+-------------+------------+----------------+----------+------------------------------------------+
|Date         | Version    | created under  | Author   | Remark                                   |
+=============+============+================+==========+==========================================+
|2022-01      | 1.0.0.0    | V3.1.4024.22   | ADBO     | Function block created                   |
+-------------+------------+----------------+----------+------------------------------------------+

*)

(* Check if any input address is different than zero*)
IF sMessageAddr <> 0 AND stSendDataAddr <> 0 THEN
	(* Access to adress*)
	psMessage := sMessageAddr;
	pstSendData := stSendDataAddr;
	
	pstSendData^.iLength := INT_TO_UDINT(LEN(psMessage^));
	
	(* Copy bytes from string to structure *)
	MEMCPY(destAddr := stSendDataAddr, srcAddr := sMessageAddr, n := pstSendData^.iLength);

	(* Function done *)
	FUN_StringToTcpBufferData := TRUE;
(* One of adresses was not correct *)
ELSE
	FUN_StringToTcpBufferData := FALSE;
END_IF

END_FUNCTION

// ---- POUs/Libs/Communication/TcpIp/FUN_TcpBufferDataToString.TcPOU
(* :Description:  This function is used to convert byte structure into string text message. Structure is recived from any TCP/IP device *)
FUNCTION FUN_TcpBufferDataToString : BOOL
VAR_INPUT
	sMessageAddr		: PVOID;						(* Destination string message *)
	stReturnDataAddr	: PVOID;						(* Source TCP/IP data structure *)
END_VAR
VAR
	psMessage			: POINTER TO STRING;			(* Pointer to string converted to structure *)
	pstReturnData		: POINTER TO ST_TcpBufferData;	(* Pointer to structure made of string bytes *)
END_VAR
(*
Version history:

+-------------+------------+----------------+----------+------------------------------------------+
|Date         | Version    | created under  | Author   | Remark                                   |
+=============+============+================+==========+==========================================+
|2022-01      | 1.0.0.0    | V3.1.4024.22   | ADBO     | Function block created                   |
+-------------+------------+----------------+----------+------------------------------------------+

*)

(* Check if any input address is different than zero*)
IF sMessageAddr <> 0 AND stReturnDataAddr <> 0 THEN
	(* Access to adress*)
	psMessage := sMessageAddr;
	pstReturnData := stReturnDataAddr;
	
	(* Clear string from any old bytes *)
	MEMSET(psMessage,0,SIZEOF(psMessage^));
	
	(* Copy bytes from string to structure *)
	MEMCPY(destAddr := psMessage, srcAddr := ADR(pstReturnData^.arrData), n:= pstReturnData^.iLength);
	
	(* Function done *)	
	FUN_TcpBufferDataToString := TRUE;
(* One of adresses was not correct *)		
ELSE
	FUN_TcpBufferDataToString := FALSE;
END_IF

END_FUNCTION

// ---- POUs/Libs/Communication/TcpIp/Tcp Buffer/FB_TcpBuffer.TcPOU
(* 
:Description: This function block represent basic TCP/IP data buffer. It is used by all TCP devices to store data to send and recive from other devices.
*)
FUNCTION_BLOCK FB_TcpBuffer

VAR CONSTANT
	iLENGTH_OF_MESSAGE		: UDINT := 8192;
	iMAX_NUMBER_OF_MESSAGES	: UDINT := 10;
END_VAR

VAR
	arrBufferMessage	: ARRAY[0..iMAX_NUMBER_OF_MESSAGES] OF ST_TcpBufferData;
	{attribute 'hide'}
	iFirstMessageIndex	: UDINT;
	{attributee 'hide'}
	iLastMessageIndex	: UDINT;
END_VAR

(* Returns TRUE if everything went fine, FALSE if buffer is full *)
METHOD MR_Append : BOOL 
VAR_INPUT
	stData	:	ST_TcpBufferData;
END_VAR
(* Clear buffer *)
IF (arrBufferMessage[iLastMessageIndex].iLength = 0) THEN
	arrBufferMessage[iLastMessageIndex] := stData;
	MR_Append := TRUE;	
	
(* Increment one index and append data to row *)
ELSIF iLastMessageIndex < iMAX_NUMBER_OF_MESSAGES THEN
	iLastMessageIndex := iLastMessageIndex + 1;
	arrBufferMessage[iLastMessageIndex] := stData;
	MR_Append := TRUE;
	
(* Start from 0 index *)
ELSIF iFirstMessageIndex > 0 THEN
	iLastMessageIndex := 0;
	arrBufferMessage[iLastMessageIndex] := stData;
	MR_Append := TRUE;

(* Buffer is full *)	
ELSE
	MR_Append := FALSE;
	
END_IF
END_METHOD

(* Clears buffer *)
METHOD MR_Clear : BOOL
VAR_INPUT
END_VAR
MEMSET(	destAddr	:=	ADR(arrBufferMessage),
		fillByte	:=	0,
		n			:=	SIZEOF(arrBufferMessage));
		
iFirstMessageIndex := 0;
iLastMessageIndex := 0;

MR_Clear := TRUE;
END_METHOD

(* Gets last data structure from buffer *)
METHOD MR_GetLast : ST_TcpBufferData
VAR_INPUT
END_VAR
MR_GetLast := arrBufferMessage[iLastMessageIndex];
END_METHOD

(* Gets last data structure from buffer and removes it*)
METHOD MR_GetNextAndRemove : ST_TcpBufferData;
VAR_INPUT
END_VAR
(*Get data *)
MR_GetNextAndRemove := arrBufferMessage[iFirstMessageIndex];

(*Remove data from index *)
MEMSET(	destAddr	:=	ADR(arrBufferMessage[iFirstMessageIndex]), 
		fillByte	:=	0, 
		n			:=	SIZEOF(arrBufferMessage[iFirstMessageIndex]));

(* Change index of first message if it's not the only message *)
IF iFirstMessageIndex <> iLastMessageIndex THEN 
	
	(* Incerment index *)
	IF iFirstMessageIndex < iMAX_NUMBER_OF_MESSAGES THEN 
		iFirstMessageIndex := iFirstMessageIndex + 1;
	
	(* End of buffer, go to 0 *)	
	ELSE 
		iFirstMessageIndex := 0;
		
	END_IF
	
END_IF
END_METHOD

END_FUNCTION_BLOCK

// ---- POUs/Libs/Communication/TcpIp/Tcp Client/FB_TcpClient.TcPOU
(* 
| :Description: This function block represent basic TCP/IP client. 
| Use MR_Init to connect to the server. 
| To send data to server use MR_AppendToSendBuffer, use FUN_StringToTcpBufferData to convert string into structure of bytes.
| If the lenght of LastRecivedMessage is bigger than 0 then you recived message from server, use FUN_TcpBufferDataToString to copy it to string message.
| To close the connection use MR_Abort.
*)
FUNCTION_BLOCK FB_TcpClient EXTENDS FB_TcpDevice
VAR		
	(* Function blocks *)
	fbSocketConnect : FB_SocketConnect;		(* FB used to connect the client to remote server *)
END_VAR
(*
Version history:

+-------------+------------+----------------+----------+-------------------------------------------------------------------------------------+
|Date         | Version    | created under  | Author   | Remark                                                                              |
+=============+============+================+==========+=====================================================================================+
|2022-01      | 1.0.0.0    | V3.1.4024.22   | ADBO     | Function block created                                                              |
+-------------+------------+----------------+----------+-------------------------------------------------------------------------------------+
|2022-02      | 1.1.0.0    | V3.1.4024.22   | ADBO     | - Added fixes to init failure reset (MS_Aborting)                                   |
|             |            |                |          | - Changed aproach in executing all FB's ( Deleted checking error before executing ) |
+-------------+------------+----------------+----------+-------------------------------------------------------------------------------------+

*)

SUPER^();

METHOD PROTECTED MS_Aborting
IF bInitFailed THEN
	fbSocketConnect( bExecute := FALSE);
	eTcpDeviceState := TCPIP_DEVICE_UNINITIALIZED;
	
ELSE
	stSocketToClose := stHSocket;
	SUPER^.MS_Aborting();
	
END_IF
END_METHOD

(* TCP/IP client is preparing to work *)
METHOD PROTECTED MS_Initializing
SUPER^.MS_Initializing();

(* Create connection socket to remote host *)
fbSocketConnect(	sSrvNetId	:= sAmsNetID,
					sRemoteHost := sHost,
					nRemotePort := iPort,
					bExecute 	:= TRUE,
					tTimeout	:= tTimeout,
					hSocket		=> stHSocket);
						
(* Socket created *)
IF NOT fbSocketConnect.bBusy AND NOT fbSocketConnect.bError THEN
	fbSocketConnect( bExecute := FALSE);
	eTcpDeviceState := TCPIP_DEVICE_READY_INITIALIZED;
	
(*Error occured while creating client socket *)
ELSIF fbSocketConnect.bError THEN
	bError := TRUE;
	iErrorID := fbSocketConnect.nErrId;
	fbAlarmCreatingClient.ipArguments.Clear().AddUDInt(iErrorID);	
	fbAlarmCreatingClient.Raise(0);
		
END_IF
END_METHOD

END_FUNCTION_BLOCK

// ---- POUs/Libs/Communication/TcpIp/Tcp Device/FB_TcpDevice.TcPOU
(* :Description: This function block represent basic TCP/IP device. It is used to build other function blocks like client and server. *)
FUNCTION_BLOCK ABSTRACT FB_TcpDevice IMPLEMENTS I_TcpDevice
VAR
	bFirstCycle 			: BOOL := TRUE;				(* First cycle bit *)		
	sName 					: STRING;					(* TCP/IP device name for other utilities *)
	
	(* Internal commadns *)
	bInit					: BOOL;						(* Initialize  TCP/IP device*)
	bAbort 					: BOOL;						(* Deinitialize TCP/IP device*)
	
	(* Internal status *)
	bActive					: BOOL;						(* TCP/IP device initialized and ready to work *)
	bBusy					: BOOL;						(* TCP/IP device is currently proccesing *)
	bError					: BOOL;						(* Error occured while executing *)
	bInitFailed				: BOOL;						(* Error occured while initializing *)
	iErrorID 				: UDINT;					(* Error ID*)
	eTcpDeviceState		 	: E_TcpIpDeviceState;		(* Current state of TCP/IP device*)
	eTcpDeviceSendState		: E_TcpIpDeviceStateSend;	(* Sending procedure state machine *)
	eTcpDeviceReciveState	: E_TcpIpDeviceStateRecive;	(* Reciving procedure state machine *)
	bConnectionLostError 	: BOOL;						(* Internal data exchange error - occured only in Running state *)

	(* Internal parameters *)
	sHost					: T_IPv4Addr;				(* IP address *)
	sAmsNetID 				: T_AmsNetID;				(* AMS network address *)
	iPort					: UINT;						(* Communication port *)
	tTimeout				: TIME;						(* Connection timeout *)
	stHSocket				: T_HSOCKET;				(* Socket handle *)
	stSocketToClose			: T_HSOCKET;

	(* Data buffers *)
	fbReceiveBuffer			: FB_TcpBuffer;				(* Custom buffer made to store recived data in bytes *)
	fbSendBuffer			: FB_TcpBuffer;				(* Custom buffer made to store send data in bytes *)
	
	(* Function blocks *)
	fbSocketClose 			: FB_SocketClose;			(* FB to close current connection*)
	fbSocketSend			: FB_SocketSend;			(* FB to send buffered data *)
	fbSocketRecive			: FB_SocketReceive;			(* FB to recive data*)
	
	(* Tc3 EventLogger - messages *)
	fbAlarmConnectionLost 		: FB_TcAlarm;			(*  *)
	fbAlarmClosingSocket		: FB_TcAlarm;			(*  *)
	fbAlarmCreatingListener	 	: FB_TcAlarm;			(*  *)
	fbAlarmCreatingClient		: FB_TcAlarm;			(*  *)
	fbAlarmClosingConnection	: FB_TcAlarm;			(*  *)
	fbAlarmWaitingForClient		: FB_TcAlarm;			(*  *)	

	bResetConfirmation 		: BOOL;						(*  *)
	
	rtError						: R_TRIG; 				(* Rising edge trigger for function block error *)
	
END_VAR
(*
Version history:

+-------------+------------+----------------+----------+-------------------------------------------------------------------------------------+
|Date         | Version    | created under  | Author   | Remark                                                                              |
+=============+============+================+==========+=====================================================================================+
|2022-01      | 1.0.0.0    | V3.1.4024.22   | ADBO     | Function block created                                                              |
+-------------+------------+----------------+----------+-------------------------------------------------------------------------------------+
|2022-02      | 1.1.0.0    | V3.1.4024.22   | ADBO     | - Added fixes to init failure reset (MS_Aborting)                                   |
|             |            |                |          | - Changed aproach in executing all FB's ( Deleted checking error before executing ) |
+-------------+------------+----------------+----------+-------------------------------------------------------------------------------------+

*)

(* First cycle procedure *)
IF bFirstCycle THEN
	bFirstCycle := FALSE;
	
	fbAlarmConnectionLost.CreateEx( stEventEntry := TC_EVENTS.ShellTcpIpDeviceEventClass.ConnectionLost, 
									bWithConfirmation := 1,
									ipSourceInfo := 0);
									
	fbAlarmClosingSocket.CreateEx( stEventEntry := TC_EVENTS.ShellTcpIpDeviceEventClass.ClosingSocket, 
									bWithConfirmation := 1,
									ipSourceInfo := 0);			
									
	fbAlarmCreatingListener.CreateEx( stEventEntry := TC_EVENTS.ShellTcpIpDeviceEventClass.CreatingListener, 
									bWithConfirmation := 1,
									ipSourceInfo := 0);			
									
	fbAlarmCreatingClient.CreateEx( stEventEntry := TC_EVENTS.ShellTcpIpDeviceEventClass.CreatingClient, 
									bWithConfirmation := 1,
									ipSourceInfo := 0);		
									
	fbAlarmClosingConnection.CreateEx( stEventEntry := TC_EVENTS.ShellTcpIpDeviceEventClass.ClosingConnection, 
									bWithConfirmation := 1,
									ipSourceInfo := 0);		
	
	fbAlarmWaitingForClient.CreateEx( stEventEntry := TC_EVENTS.ShellTcpIpDeviceEventClass.WaitingForClient, 
									bWithConfirmation := 1,
									ipSourceInfo := 0);		
									
END_IF

(* Report errors that occur *)
rtError(CLK:=bError);

IF rtError.Q THEN 
	fbMachineLogger.MR_AddLogs(FUN_MergeStrings5(sName, ' : Error occured (error ID: ', UDINT_TO_STRING(iErrorID), ')', ''));

END_IF

(* Execute state machine *)
StateMachine();

(* Active status bit control*)
bActive := eTcpDeviceState = TCPIP_DEVICE_RUNNING OR eTcpDeviceState = TCPIP_DEVICE_ABORTING;

PROPERTY Active : REFERENCE TO BOOL
GET
Active REF= bActive;
END_GET
END_PROPERTY

PROPERTY AmsNetId : T_IPv4Addr
GET
AmsNetId := sAmsNetID;
END_GET
SET
sAmsNetID := AmsNetId;
END_SET
END_PROPERTY

PROPERTY Error : REFERENCE TO BOOL
GET
Error REF= bError;
END_GET
END_PROPERTY

PROPERTY ErrorID : REFERENCE TO UDINT
GET
ErrorID REF= iErrorID;
END_GET
END_PROPERTY

PROPERTY Host : T_IPv4Addr
GET
Host := sHost;
END_GET
SET
sHost := Host;
END_SET
END_PROPERTY

PROPERTY LastRecivedMessage : ST_TcpBufferData
GET
(*
stLastRecivedMessageTemp := fbReceiveBuffer.MR_GetLast();
LastRecivedMessage REF= stLastRecivedMessageTemp;
*)
LastRecivedMessage := fbReceiveBuffer.MR_GetLast();
END_GET
END_PROPERTY

(* Abort connection and go back to uninitialized state *)
METHOD MR_Abort : BOOL
VAR_INPUT
END_VAR
IF eTcpDeviceState > TCPIP_DEVICE_UNINITIALIZED THEN
	bAbort := TRUE;
	bInit := FALSE;
	bInitFailed := eTcpDeviceState = TCPIP_DEVICE_INITIALIZING;	
	eTcpDeviceState := TCPIP_DEVICE_ABORTING;
	fbMachineLogger.MR_AddLogs(CONCAT(sName,' : abort requested'));
	
ELSIF eTcpDeviceState = TCPIP_DEVICE_UNINITIALIZED THEN
	bAbort := FALSE;
	bInitFailed := FALSE;
	MR_Abort := TRUE;
	fbMachineLogger.MR_AddLogs(CONCAT(sName,' : abort done'));
	
END_IF
END_METHOD

(* Add data to send buffer *)
METHOD MR_AppendToSendBuffer : BOOL
VAR_INPUT
	stData : ST_TcpBufferData;
END_VAR
IF eTcpDeviceState = TCPIP_DEVICE_RUNNING THEN
	MR_AppendToSendBuffer := fbSendBuffer.MR_Append(stData);
END_IF
END_METHOD

(* Clear intearnal send and recive buffer *)
METHOD MR_ClearAllBuffers : BOOL
VAR_INPUT
END_VAR
MR_ClearAllBuffers := fbSendBuffer.MR_Clear() AND fbReceiveBuffer.MR_Clear();
END_METHOD

METHOD MR_ClearReciveBuffer : BOOL
VAR_INPUT
END_VAR
MR_ClearReciveBuffer := fbReceiveBuffer.MR_Clear();
END_METHOD

METHOD MR_ClearSendBuffer : BOOL
VAR_INPUT
END_VAR
MR_ClearSendBuffer := fbSendBuffer.MR_Clear();
END_METHOD

(* Set the initial parameters of TCP/IP device *)
METHOD MR_FirstCycle : BOOL
VAR_INPUT
	sName 		: STRING;		(* TCP/IP Device name for identyfication *)
	sHost		: T_IPv4Addr;	(* TCP/IP-Client: IP address of remote server/ TCP/IP-Server: local server IP address *)
	sAmsNetID	: T_AmsNetID;	(* TCP/IP-Client: AMS network address of remote server/ TCP/IP-Server: local server ams network address *)
	iPort		: UINT;			(* TCP/IP-Client: Port of remote server/ TCP/IP-Server: local server port *)
	tTimeout	: TIME;			(* Connection timeout *)
END_VAR
THIS^.sName 	:= sName;
THIS^.sHost 	:= sHost;
THIS^.sAmsNetID := sAmsNetID;
THIS^.iPort 	:= iPort;
THIS^.tTimeout 	:= tTimeout;
END_METHOD

(* Start initialization of TCP/IP device *)
METHOD MR_Init : BOOL
VAR_INPUT
END_VAR
IF eTcpDeviceState = TCPIP_DEVICE_UNINITIALIZED THEN
	bInit := TRUE;
	eTcpDeviceState := TCPIP_DEVICE_INITIALIZING;
	fbMachineLogger.MR_AddLogs(CONCAT(sName,' : initialization requested'));
		
ELSIF eTcpDeviceState = TCPIP_DEVICE_RUNNING THEN
	bInit := FALSE;
	MR_Init := TRUE;
	fbMachineLogger.MR_AddLogs(CONCAT(sName,' : initialization done'));	
	
END_IF
END_METHOD

(* TCP/IP device is reseting to uninitialized mode*)
METHOD PROTECTED MS_Aborting
(* Close current conncetion socket *)
fbSocketClose(	sSrvNetId 	:= sAmsNetID,
				hSocket		:= stSocketToClose,
				bExecute	:= TRUE,
				tTimeout	:= DEFAULT_ADS_TIMEOUT);
	
(* Socket closed *)				
IF NOT fbSocketClose.bBusy AND NOT fbSocketClose.bError THEN
	eTcpDeviceState := TCPIP_DEVICE_UNINITIALIZED;
	
(* Error occured while closing the socket *)
ELSIF fbSocketClose.bError THEN
	bError := TRUE;
	iErrorID := fbSocketClose.nErrId;
	fbAlarmClosingSocket.ipArguments.Clear().AddUDInt(iErrorID);	
	fbAlarmClosingSocket.Raise(0);
	
END_IF
END_METHOD

(* TCP/IP device is preparing to work *)
METHOD PROTECTED MS_Initializing
eTcpDeviceSendState := TCPIP_DEVICE_DATA_EXCHANGE_GET_SEND_DATA;
eTcpDeviceReciveState := TCPIP_DEVICE_DATA_EXCHANGE_GET_RECIVED_DATA;
END_METHOD

(* TCP/IP device is ready to work *)
METHOD PROTECTED MS_ReadyInitialized
(* Skip to device running state *)
eTcpDeviceState := TCPIP_DEVICE_RUNNING;
END_METHOD

(* TCP/IP device is working in the network *)
METHOD PROTECTED MS_Running
VAR_INST
	stDataToSend		:	ST_TcpBufferData;			(* Data to send structure *)
	stReceivedData		:	ST_TcpBufferData;			(* Recived data structure *)
	bRepeatLoop			:	BOOL;						(* Loop control bit *)
END_VAR
IF NOT bConnectionLostError THEN
	(* Send data loop *)
	REPEAT
		bRepeatLoop := FALSE;
	
		CASE eTcpDeviceSendState OF
			(*Get data to send from buffer *)
			TCPIP_DEVICE_DATA_EXCHANGE_GET_SEND_DATA:
				stDataToSend := fbSendBuffer.MR_GetNextAndRemove();
				IF stDataToSend.iLength > 0 THEN
					eTcpDeviceSendState := TCPIP_DEVICE_DATA_EXCHANGE_SEND;
					bRepeatLoop := TRUE;
					
				END_IF
			
			TCPIP_DEVICE_DATA_EXCHANGE_SEND:
				(*Send buffered data to host*)
				fbSocketSend(	sSrvNetID 	:= sAmsNetID,
								hSocket		:= stHSocket,
								cbLen		:= stDataToSend.iLength,
								pSrc		:= ADR(stDataToSend.arrData),
								bExecute	:= TRUE);
				
				eTcpDeviceSendState := TCPIP_DEVICE_DATA_EXCHANGE_SEND_DONE;
				bRepeatLoop := TRUE;
				
			TCPIP_DEVICE_DATA_EXCHANGE_SEND_DONE:	
				(* Sending done go get next data row *)			
				IF NOT fbSocketSend.bBusy AND NOT fbSocketSend.bError THEN
					fbSocketSend(bExecute := FALSE );
					eTcpDeviceSendState := TCPIP_DEVICE_DATA_EXCHANGE_GET_SEND_DATA;
					bRepeatLoop := TRUE;
						
				(* Sending in progress *)
				ELSIF fbSocketSend.bBusy AND NOT fbSocketSend.bError THEN
					eTcpDeviceSendState := TCPIP_DEVICE_DATA_EXCHANGE_SEND;
					
				(* Error occured while sending the data *)
				ELSIF fbSocketSend.bError THEN
					bError := TRUE;
					iErrorID := fbSocketSend.nErrId;
					bConnectionLostError := TRUE;
					fbAlarmConnectionLost.ipArguments.Clear().AddUDInt(iErrorID);	
					fbAlarmConnectionLost.Raise(0);
					
				END_IF
		END_CASE
	UNTIL 
		NOT bRepeatLoop
	END_REPEAT
ELSE
	fbSocketSend( bExecute := FALSE);
	
END_IF

IF NOT bConnectionLostError THEN
	(* Recive data loop *)
	REPEAT
		bRepeatLoop := FALSE;
		
		CASE eTcpDeviceReciveState OF
			TCPIP_DEVICE_DATA_EXCHANGE_GET_RECIVED_DATA:
				fbSocketRecive( 	sSrvNetId	:=	sAmsNetID,
									hSocket		:=	stHSocket,
									cbLen		:=	SIZEOF(stReceivedData.arrData),
									pDest		:=	ADR(stReceivedData.arrData),
									bExecute	:=	TRUE);
			
			eTcpDeviceReciveState := TCPIP_DEVICE_DATA_EXCHANGE_RECIVE_DONE;
			bRepeatLoop := TRUE;
			
			TCPIP_DEVICE_DATA_EXCHANGE_RECIVE_DONE:		
				IF NOT fbSocketRecive.bBusy AND NOT fbSocketRecive.bError THEN
					stReceivedData.iLength	:=	fbSocketRecive.nRecBytes;
					fbSocketRecive(	bExecute := FALSE );
					eTcpDeviceReciveState := TCPIP_DEVICE_DATA_EXCHANGE_WRITE_TO_BUFFER;
					bRepeatLoop := TRUE;
					
				ELSIF fbSocketRecive.bBusy AND NOT fbSocketRecive.bError THEN
					eTcpDeviceReciveState := TCPIP_DEVICE_DATA_EXCHANGE_GET_RECIVED_DATA;
					bRepeatLoop := FALSE;		
	
				ELSIF fbSocketRecive.bError THEN
					bError := TRUE;
					iErrorID := fbSocketRecive.nErrId;
					bConnectionLostError := TRUE;
					fbAlarmConnectionLost.ipArguments.Clear().AddUDInt(iErrorID);
					fbAlarmConnectionLost.Raise(0);
					eTcpDeviceReciveState := TCPIP_DEVICE_DATA_EXCHANGE_GET_RECIVED_DATA;
					
				END_IF
			
			TCPIP_DEVICE_DATA_EXCHANGE_WRITE_TO_BUFFER: // write data to buffer
				IF stReceivedData.iLength > 0 THEN
					fbReceiveBuffer.MR_Append(stReceivedData);
					
				END_IF
					eTcpDeviceReciveState := TCPIP_DEVICE_DATA_EXCHANGE_GET_RECIVED_DATA;
					bRepeatLoop := TRUE;
			
		END_CASE
	UNTIL 
		NOT bRepeatLoop
		
	END_REPEAT
ELSE
	fbSocketRecive(bExecute := FALSE);	
	
END_IF
END_METHOD

(* TCP/IP device is not ready to work *)
METHOD PROTECTED MS_Uninitialized
(* Reseting common function blocks *)
fbSocketSend( bExecute := FALSE);
fbSocketRecive( bExecute := FALSE);
fbSocketClose( bExecute := FALSE);

(* Clearing buffers *)
fbReceiveBuffer.MR_Clear();
fbSendBuffer.MR_Clear();

(* Reseting flags and error codes *)
bActive 				:= FALSE;
bBusy 					:= FALSE;
bError 					:= FALSE;
bInitFailed				:= FALSE;
bConnectionLostError	:= FALSE;
iErrorID 				:= 0;

(* Confirming and resetting alarms *)
fbAlarmConnectionLost.Confirm( nTimeStamp := 0);
fbAlarmClosingSocket.Confirm( nTimeStamp := 0);
fbAlarmCreatingListener.Confirm( nTimeStamp := 0);
fbAlarmCreatingClient.Confirm( nTimeStamp := 0);
fbAlarmClosingConnection.Confirm( nTimeStamp := 0);
fbAlarmWaitingForClient.Confirm( nTimeStamp := 0);

fbAlarmConnectionLost.Clear( nTimeStamp := 0, bResetConfirmation := bResetConfirmation); 
fbAlarmClosingSocket.Clear( nTimeStamp := 0, bResetConfirmation := bResetConfirmation); 
fbAlarmCreatingListener.Clear( nTimeStamp := 0, bResetConfirmation := bResetConfirmation); 
fbAlarmCreatingClient.Clear( nTimeStamp := 0, bResetConfirmation := bResetConfirmation); 
fbAlarmClosingConnection.Clear( nTimeStamp := 0, bResetConfirmation := bResetConfirmation); 
fbAlarmWaitingForClient.Clear( nTimeStamp := 0, bResetConfirmation := bResetConfirmation);
END_METHOD

PROPERTY NextRecivedMessage : ST_TcpBufferData
GET
(*
stNextRecivedMessageTemp := fbReceiveBuffer.MR_GetNextAndRemove();
NextRecivedMessage REF= stNextRecivedMessageTemp;
*)
NextRecivedMessage := fbReceiveBuffer.MR_GetNextAndRemove();
END_GET
END_PROPERTY

PROPERTY Port : UINT
GET
Port := iPort;
END_GET
SET
iPort := Port;
END_SET
END_PROPERTY

PROPERTY State : REFERENCE TO E_TcpIpDeviceState
GET
State REF= eTcpDeviceState;
END_GET
END_PROPERTY

(* Standard state machine call for TCP/IP device *)
METHOD PROTECTED StateMachine
CASE eTcpDeviceState OF
	(* TCP/IP device is not ready to work *)
	TCPIP_DEVICE_UNINITIALIZED:
		MS_Uninitialized();
	
	(* TCP/IP device is preparing to work *)	
	TCPIP_DEVICE_INITIALIZING:
		MS_Initializing();
	
	(* TCP/IP device is ready to work *)	
	TCPIP_DEVICE_READY_INITIALIZED:
		MS_ReadyInitialized();
		
	(* TCP/IP device is working in the network *)
	TCPIP_DEVICE_RUNNING:
		MS_Running();
	
	(* TCP/IP device is reseting to uninitialized mode*)	
	TCPIP_DEVICE_ABORTING:
		MS_Aborting();
		
END_CASE
END_METHOD

PROPERTY Timeout : TIME
GET
Timeout := tTimeout;
END_GET
SET
tTimeout := Timeout;
END_SET
END_PROPERTY

END_FUNCTION_BLOCK

// ---- POUs/Libs/Communication/TcpIp/Tcp Server/FB_TcpServer.TcPOU
(* 
:Description: This function block represent basic TCP/IP client.
*)
FUNCTION_BLOCK FB_TcpServer EXTENDS FB_TcpDevice
VAR
	(* Internal command *)
	bDisconnect			: BOOL := FALSE;		(* Disconnect server from current connection *)	
	
	(* Internal parameters *)
	stHListener			: T_HSOCKET;			(* Server listener handle *)
	
	(* Internal status *)
	eTcpServerState		: E_TcpIpServerStateRunning;	(* Current server state while running *)
	
	(* Function blocks*)
	fbSocketAccept		: FB_SocketAccept;		(* FB to listen for clienncts connection requests *)
	fbSocketListen		: FB_SocketListen;		(* FB create servers listener socket *)
	
END_VAR
(*
Version history:

+-------------+------------+----------------+----------+-------------------------------------------------------------------------------------+
|Date         | Version    | created under  | Author   | Remark                                                                              |
+=============+============+================+==========+=====================================================================================+
|2022-01      | 1.0.0.0    | V3.1.4024.22   | ADBO     | Function block created                                                              |
+-------------+------------+----------------+----------+-------------------------------------------------------------------------------------+
|2022-02      | 1.1.0.0    | V3.1.4024.22   | ADBO     | - Added fixes to init failure reset (MS_Aborting)                                   |
|             |            |                |          | - Changed aproach in executing all FB's ( Deleted checking error before executing ) |
+-------------+------------+----------------+----------+-------------------------------------------------------------------------------------+
|2022-02      | 1.1.1.0    | V3.1.4024.22   | ADBO     | - Fixed bug when MR_Disconect stucked before switch to connection closing state     |
+-------------+------------+----------------+----------+-------------------------------------------------------------------------------------+

*)

SUPER^();

(* Stop connection with current client and wait for another connection *)
METHOD MR_Disconnect : BOOL
VAR_INPUT
END_VAR
IF eTcpDeviceState = TCPIP_DEVICE_RUNNING AND eTcpServerState = TCPIP_SERVER_RUNNING_DATA_EXCHANGE THEN
	bDisconnect := TRUE;
	fbMachineLogger.MR_AddLogs(CONCAT(sName,' : disconnection requested'));

ELSIF eTcpDeviceState = TCPIP_DEVICE_RUNNING AND eTcpServerState = TCPIP_SERVER_RUNNING_CLOSE_CONNECTION_DONE THEN
	bDisconnect := FALSE;
	MR_Disconnect := TRUE;
	fbMachineLogger.MR_AddLogs(CONCAT(sName,' : disconnection done'));
END_IF
END_METHOD

METHOD PROTECTED MS_Aborting
IF bInitFailed THEN
	fbSocketListen( bExecute := FALSE);
	fbSocketAccept( bExecute := FALSE);
	eTcpDeviceState := TCPIP_DEVICE_UNINITIALIZED;
	
ELSE
	stSocketToClose := stHListener;
	SUPER^.MS_Aborting();
	
END_IF
END_METHOD

(* TCP/IP server is preparing to work *)
METHOD PROTECTED MS_Initializing
SUPER^.MS_Initializing();

(* Creating server listener socket at selected address and port *)
fbSocketListen( sSrvNetId	:= sAmsNetID,
				sLocalHost	:= sHost,
				nLocalPort	:= iPort,
				bExecute	:= TRUE,
				tTimeout	:= DEFAULT_ADS_TIMEOUT,
				hListener	=> stHListener);
					
(* Socket created *)	
IF NOT fbSocketListen.bBusy AND NOT fbSocketListen.bError THEN
	fbSocketListen( bExecute := FALSE);
	eTcpDeviceState := TCPIP_DEVICE_READY_INITIALIZED;
	eTcpServerState := TCPIP_SERVER_RUNNING_START_LISTENING;
		
(* Error occured while creating listener socket *)
ELSIF fbSocketListen.bError THEN	
	bError := TRUE;
	iErrorID := fbSocketListen.nErrId;
	fbAlarmCreatingListener.ipArguments.Clear().AddUDInt(iErrorID);	
	fbAlarmCreatingListener.Raise(0);
	
END_IF
END_METHOD

METHOD PROTECTED MS_Running
VAR_INST
	stDataToSend	:	ST_TcpBufferData;			(* Data to send structure *)
	stReceivedData	:	ST_TcpBufferData;			(* Recived data structure *)
	bRepeatLoop		:	BOOL;						(* Loop control bit *)
END_VAR
CASE eTcpServerState OF
	(* Reset listening FB*)
	TCPIP_SERVER_RUNNING_START_LISTENING:
		fbSocketAccept( bExecute := FALSE);
		eTcpServerState := TCPIP_SERVER_RUNNING_WAIT_FOR_CONNECTION;
	
	(* Wait for client connection *)
	TCPIP_SERVER_RUNNING_WAIT_FOR_CONNECTION:
		fbSocketAccept( sSrvNetId	:= sAmsNetID,
						hListener	:= stHListener,
						bExecute	:= TRUE,
						tTimeout	:= tTimeout);
			
		(* FB finished work without error *)			
		IF NOT fbSocketAccept.bBusy AND NOT fbSocketAccept.bError THEN
			(* Client connected *)
			IF fbSocketAccept.bAccepted THEN
				stHSocket := fbSocketAccept.hSocket;
				fbSocketAccept( bExecute := FALSE);
				
				eTcpDeviceSendState := TCPIP_DEVICE_DATA_EXCHANGE_GET_SEND_DATA;
				eTcpDeviceReciveState := TCPIP_DEVICE_DATA_EXCHANGE_GET_RECIVED_DATA;
				eTcpServerState := TCPIP_SERVER_RUNNING_DATA_EXCHANGE;
				fbMachineLogger.MR_AddLogs(CONCAT(sName,' : client connected'));
			
				(* Client not connected *)
			ELSE
				eTcpServerState := TCPIP_SERVER_RUNNING_START_LISTENING;
				
			END_IF
			
		(* Error occured while waiting for connection *)	
		ELSIF fbSocketAccept.bError THEN
			bError := TRUE;
			iErrorID := fbSocketAccept.nErrId;
			fbAlarmWaitingForClient.ipArguments.Clear().AddUDInt(iErrorID);	
			fbAlarmWaitingForClient.Raise(0);
			
		END_IF
			
	
	TCPIP_SERVER_RUNNING_DATA_EXCHANGE:
		(* Safe end of data exchange - disconnect from current connection *)
		IF bDisconnect THEN
			fbReceiveBuffer.MR_Clear();
			fbSendBuffer.MR_Clear();
			fbSocketSend(bExecute := FALSE);
			fbSocketRecive(bExecute := FALSE);
			
			IF NOT fbSocketSend.bBusy AND NOT fbSocketRecive.bBusy THEN
				eTcpServerState := TCPIP_SERVER_RUNNING_CLOSE_CONNECTION;
				
			END_IF
			
		(* Standard data exchange procedure *)
		ELSE
			SUPER^.MS_Running(); 
			
		END_IF	
	
	TCPIP_SERVER_RUNNING_CLOSE_CONNECTION:
		(* Close current connection *)
		fbSocketClose( 	sSrvNetId 	:= sAmsNetID,
						hSocket		:= stHSocket,
						bExecute	:= TRUE,
						tTimeout	:= tTimeout);
			
		(* Connection closed *)
		IF NOT fbSocketClose.bBusy AND NOT fbSocketClose.bError THEN
			fbSocketClose( bExecute := FALSE);
			eTcpServerState := TCPIP_SERVER_RUNNING_CLOSE_CONNECTION_DONE;
			
		(* Error occured while closing the connection *)
		ELSIF fbSocketClose.bError THEN
			bError := TRUE;
			iErrorID := fbSocketClose.nErrId;
			fbAlarmClosingConnection.ipArguments.Clear().AddUDInt(iErrorID);	
			fbAlarmClosingConnection.Raise(0);
			
		END_IF
	
	TCPIP_SERVER_RUNNING_CLOSE_CONNECTION_DONE:
		(* Disconnect procedure done *)
		IF NOT bDisconnect THEN
			fbSocketSend( bExecute := FALSE);
			fbSocketRecive( bExecute := FALSE);
			bError := FALSE;
			iErrorID := 0;
			bConnectionLostError := FALSE;
			eTcpServerState := TCPIP_SERVER_RUNNING_START_LISTENING;
			
		END_IF	
	
END_CASE
END_METHOD

PROPERTY ServerState : REFERENCE TO E_TcpIpServerStateRunning
GET
ServerState REF= eTcpServerState;
END_GET
END_PROPERTY

END_FUNCTION_BLOCK

// ---- POUs/Libs/Cylinder/Double Coil Cylinder/FB_DoubleCoilCylinder.TcPOU
FUNCTION_BLOCK FB_DoubleCoilCylinder EXTENDS FB_SingleCoilCylinder
VAR_INPUT
END_VAR
VAR_OUTPUT
END_VAR
VAR
	(* Coils *)
	poHomeValve	: FB_DigitalOutput;	(* Home position valve function block *)
END_VAR

IF bFirstCycle THEN
	poActiveValve.MR_FirstCycle( sName := CONCAT(sName,':Home_Valve'),sModuleType := ref_poHomeValve.ModuleType, sPortID := ref_poHomeValve.PortID);	
END_IF

SUPER^();

bPositionHold := poActiveValve.Out OR poHomeValve.Out;

poHomeValve();

METHOD PROTECTED MS_GoActive
VAR_INPUT
END_VAR
poHomeValve.Out := FALSE;
SUPER^.MS_GoActive();
END_METHOD

METHOD PROTECTED MS_GoHome
VAR_INPUT
END_VAR
poHomeValve.Out := TRUE;
SUPER^.MS_GoHome();
END_METHOD

METHOD PROTECTED MS_Release
VAR_INPUT
END_VAR
poHomeValve.Out := FALSE;
SUPER^.MS_Release();
END_METHOD

METHOD PROTECTED MS_Reset
VAR_INPUT
END_VAR
poHomeValve.Out := FALSE;

SUPER^.MS_Reset();
END_METHOD

METHOD PROTECTED MS_Uninitialized
poHomeValve.Out := FALSE;
SUPER^.MS_Uninitialized();
END_METHOD

PROPERTY ref_poHomeValve : REFERENCE TO FB_DigitalOutput
GET
ref_poHomeValve REF= poHomeValve;
END_GET
END_PROPERTY

END_FUNCTION_BLOCK

// ---- POUs/Libs/Cylinder/Single Coil Cylinder/FB_SingleCoilCylinder.TcPOU
FUNCTION_BLOCK FB_SingleCoilCylinder EXTENDS FB_UniversalCylinder
VAR_INPUT
	
END_VAR
VAR_OUTPUT
END_VAR
VAR
	(* Coils *)
	poActiveValve	: FB_DigitalOutput;	(* Active position valve function block *)
END_VAR

IF bFirstCycle THEN
	poActiveValve.MR_FirstCycle( sName := CONCAT(sName,':Active_Valve'),sModuleType := ref_poActiveValve.ModuleType, sPortID:= ref_poActiveValve.PortID);
END_IF

SUPER^();

bPositionHold := poActiveValve.Out;

poActiveValve();

METHOD PROTECTED M_SimulationLogic
VAR_INPUT
END_VAR
IF poActiveValve.Out THEN
	piActiveSensor.MR_SetForceValue();
	piHomeSensor.MR_ResetForceValue();
	
ELSIF NOT poActiveValve.Out THEN
	piActiveSensor.MR_ResetForceValue();
	piHomeSensor.MR_SetForceValue();
	
END_IF
END_METHOD

METHOD PROTECTED MS_GoActive
VAR_INPUT
END_VAR
poActiveValve.Out := TRUE;

CASE eCylinderGoActiveState OF
	CYLINDER_MOVE_START_TRACKING:
		piActiveSensor.MR_StartTracking();
		
		IF piActiveSensor.In THEN
			IF TIME_TO_INT(tDelay) = 0 THEN
				eCylinderGoActiveState := CYLINDER_MOVE_DONE;
			ELSE
				eCylinderGoActiveState := CYLINDER_MOVE_DELAY;
			END_IF
		END_IF
		
	CYLINDER_MOVE_DELAY:
		tonGoActiveDelay( IN := TRUE, PT := tDelay);
		
		IF tonGoActiveDelay.Q THEN
			tonGoActiveDelay( IN := FALSE );
			eCylinderGoActiveState := CYLINDER_MOVE_DONE;
		END_IF
		
	CYLINDER_MOVE_DONE:
		eCylinderState := CYLINDER_GO_ACTIVE_DONE;
		
END_CASE
END_METHOD

METHOD PROTECTED MS_GoHome
VAR_INPUT
END_VAR
poActiveValve.Out := FALSE;

CASE eCylinderGoHomeState OF
	CYLINDER_MOVE_START_TRACKING:
		piHomeSensor.MR_StartTracking();
		
		IF piHomeSensor.In THEN
			IF TIME_TO_INT(tDelay) = 0 THEN
				eCylinderGoHomeState := CYLINDER_MOVE_DONE;
			ELSE
				eCylinderGoHomeState := CYLINDER_MOVE_DELAY;
			END_IF
		END_IF
		
	CYLINDER_MOVE_DELAY:
		tonGoHomeDelay( IN := TRUE, PT := tDelay);
		
		IF tonGoHomeDelay.Q THEN
			tonGoHomeDelay( IN := FALSE);
			eCylinderGoHomeState := CYLINDER_MOVE_DONE;
		END_IF
		
	CYLINDER_MOVE_DONE:
		eCylinderState := CYLINDER_GO_HOME_DONE;
	
END_CASE
END_METHOD

METHOD PROTECTED MS_Release
VAR_INPUT
END_VAR
poActiveValve.Out := FALSE;
eCylinderState := CYLINDER_RELEASE_DONE;
END_METHOD

METHOD PROTECTED MS_Reset
VAR_INPUT
END_VAR
poActiveValve.Out := FALSE;

SUPER^.MS_Reset();
END_METHOD

METHOD PROTECTED MS_Uninitialized
poActiveValve.Out := FALSE;
SUPER^.MS_Uninitialized();
END_METHOD

PROPERTY ref_poActiveValve : REFERENCE TO FB_DigitalOutput
GET
ref_poActiveValve REF= poActiveValve;
END_GET
END_PROPERTY

END_FUNCTION_BLOCK

// ---- POUs/Libs/Cylinder/Universal Cylinder/FB_UniversalCylinder.TcPOU
(* 
:Description: This function block is used represent basic cylinder device.
*)
FUNCTION_BLOCK ABSTRACT FB_UniversalCylinder IMPLEMENTS I_UniversalCylinder
VAR
	bFirstCycle			: BOOL := TRUE;			(* First cycle procedure bit *)
	sName				: STRING;				(*  *)
	
	(* Internal commands *)
	bInit 				: BOOL;					(* Prepare cylinder to work *)
	bGoActive 			: BOOL;					(* Move cylinder to active postion *)
	bGoHome 			: BOOL;					(* Move cylinder to home postion *)
	bRelease			: BOOL;					(* Release cylinder *)
	bReset				: BOOL;					(* Reset function block *)
	bAbort				: BOOL;					(* Deinitialize function block *)
	bSimulation			: BOOL;					(* Simulation on/off bit *)
	
	(* Cylinder state *)
	bActive				: BOOL;					(*  *)
	bBusy				: BOOL;					(*  *)	
	bError 				: BOOL;					(*  *)
	bPositionActive		: BOOL;					(*  *)
	bPositionHome		: BOOL;					(*  *)
	bPositionHold		: BOOL;					(*  *)
	eErrorID 			: E_CylinderError;		(*  *)
	eCylinderState		: E_CylinderState;		(* State machine of function block *)
	eCylinderGoHomeState : E_CylinderStateGo;
	eCylinderGoActiveState : E_CylinderStateGo;
	
	(* Sensors *)
	piActiveSensor		: FB_DigitalInputExt;	(* Active position sensor function block *)
	piHomeSensor		: FB_DigitalInputExt;	(* Home position sensor function block *)
	
	(* Timers *)
	tonGoHomeDelay		: TON;					(* Timer on delay when moving to home position *)
	tonGoActiveDelay	: TON;					(* Timer on delay when moving to active position *)
	tonMeasurementTimer	: TON;					(* Measurement of movement time *)
	tonCylinderWatchdog	: TON;					(* Movement watchdog *)
	
	(* Time parameters *)
	tDelay				: TIME := T#100MS;		(* Delay time when moving to any position *)
	tMeasurement		: TIME := T#60S;		(* Time of movement measurement *)

	tMoveActive			: TIME;					(* Time of last movement to active postion *)
	tMoveHome			: TIME;					(* Time of last movement to home position *)
END_VAR
(*
Version history:

+-------------+------------+----------------+----------+------------------------------------------------------------+
|Date         | Version    | created under  | Author   | Remark                                                     |
+=============+============+================+==========+============================================================+
|2021-11      | 1.0.0.0    | V3.1.4024.22   | ADBO     | Function block created                                     |
+-------------+------------+----------------+----------+------------------------------------------------------------+
|2022-01      | 1.1.0.0    | V3.1.4024.22   | ADBO     | Function block changed into base for FB_SingleCoilCylinder |
+-------------+------------+----------------+----------+------------------------------------------------------------+
|2022-03      | 1.2.0.0    | V3.1.4024.22   | ADBO     | Changed FB_DigitalInput to FB_DigitalInputExt              |
+-------------+------------+----------------+----------+------------------------------------------------------------+

*)

(* Initial assignaments *)
IF bFirstCycle THEN
	bFirstCycle := FALSE;
	
	piHomeSensor.EnableTimeout := TRUE;
	piActiveSensor.EnableTimeout := TRUE;
END_IF

(* Simulation enabled*)
IF bSimulation THEN
	piHomeSensor.EnableForce := TRUE;
	piActiveSensor.EnableForce := TRUE;
	
	M_SimulationLogic();
ELSE
	piHomeSensor.MR_ResetForceValue();
	piActiveSensor.MR_ResetForceValue();
	piHomeSensor.EnableForce := FALSE;
	piActiveSensor.EnableForce := FALSE;
END_IF

(* Time  measurement - to active position *)
IF piActiveSensor.RisingTrigger AND eCylinderState = CYLINDER_GO_ACTIVE THEN
	tMoveActive := tonMeasurementTimer.ET;
END_IF

(* Time measurement - to home position *)
IF piHomeSensor.RisingTrigger AND eCylinderState = CYLINDER_GO_HOME THEN
	tMoveHome := tonMeasurementTimer.ET;
END_IF

(*  *)
tonMeasurementTimer(	IN := tonCylinderWatchdog.IN,
						PT := tMeasurement);

(* State machine - old *)
StateMachine();

(* Update status flags *)
bActive := eCylinderState >= CYLINDER_IDLE OR eCylinderState = CYLINDER_ABORTING ;
//bBusy := eCylinderState > CYLINDER_IDLE;
bError := piHomeSensor.ErrorTimedout OR piActiveSensor.ErrorTimedout;

(* Error handling *)
IF piHomeSensor.ErrorTimedout THEN
	eErrorID := CYLINDER_ERROR_MOVE_HOME_TIMED_OUT;
	fbMachineLogger.MR_AddLogs(FUN_MergeStrings5(sName,' : Error occured (error ID: ', 'move home timed out', ')', ''));

ELSIF piActiveSensor.ErrorTimedout THEN
	eErrorID := CYLINDER_ERROR_MOVE_ACTIVE_TIMED_OUT;
	fbMachineLogger.MR_AddLogs(FUN_MergeStrings5(sName,' : Error occured (error ID: ', 'move active timed out', ')', ''));

ELSE
	eErrorID := CYLINDER_ERROR_OK;
	
END_IF

(* Position flag update *)
bPositionActive := piActiveSensor.In;
bPositionHome := piHomeSensor.In;

(* State machine *)
//StateMachine();

(* Run sensors instances *)
piHomeSensor();
piActiveSensor();

PROPERTY Active : REFERENCE TO BOOL
GET
Active REF= bActive;
END_GET
END_PROPERTY

PROPERTY ActiveTimeout : TIME
GET
ActiveTimeout := piActiveSensor.Timeout;
END_GET
SET
piActiveSensor.Timeout := ActiveTimeout;
END_SET
END_PROPERTY

PROPERTY Busy : REFERENCE TO BOOL
GET
Busy REF= bBusy;
END_GET
END_PROPERTY

PROPERTY Delay : TIME
GET
Delay := tDelay;
END_GET
SET
tDelay := Delay;
END_SET
END_PROPERTY

PROPERTY Error : REFERENCE TO BOOL
GET
Error REF= bError;
END_GET
END_PROPERTY

PROPERTY ErrorID : REFERENCE TO E_CylinderError
GET
ErrorID REF= eErrorID;
END_GET
END_PROPERTY

PROPERTY HomeTimeout : TIME
GET
HomeTimeout := piHomeSensor.Timeout;
END_GET
SET
piHomeSensor.Timeout := HomeTimeout;
END_SET
END_PROPERTY

METHOD PROTECTED ABSTRACT M_SimulationLogic
VAR_INPUT
END_VAR
END_METHOD

PROPERTY MoveActiveTime : REFERENCE TO TIME
GET
MoveActiveTime REF= tMoveActive;
END_GET
END_PROPERTY

PROPERTY MoveHomeTime : REFERENCE TO TIME
GET
MoveHomeTime REF= tMoveHome;
END_GET
END_PROPERTY

METHOD MR_Abort : BOOL
VAR_INPUT
END_VAR
IF eCylinderState >= CYLINDER_IDLE THEN
	bBusy := TRUE;
	bAbort := TRUE;
	MR_Abort := FALSE;
	eCylinderState := CYLINDER_ABORTING;
	fbMachineLogger.MR_AddLogs(CONCAT(sName,' : abort requested'));	
	
ELSIF eCylinderState = CYLINDER_UNINITIALIZED THEN
	bAbort := FALSE;
	MR_Abort := TRUE;
	fbMachineLogger.MR_AddLogs(CONCAT(sName,' : abort done'));	
	
END_IF
END_METHOD

METHOD MR_FirstCycle : BOOL
VAR_INPUT
	sName 							: STRING;
	sHomeSensorModuleType			: STRING;
	sHomeSensorPortID				: STRING;
	sActiveSensorModuleType			: STRING;
	sActiveSensorPortID				: STRING;
	tGoHomeTimeout					: TIME;
	tGoActiveTimeout				: TIME;
	tDelay							: TIME;
END_VAR
THIS^.sName := sName;								
THIS^.tDelay := tDelay;

THIS^.piHomeSensor.MR_FirstCycleEx( sName			:= CONCAT(sName,':Home_Sensor'),
									sModuleType 	:= sHomeSensorModuleType,
									sPortID			:= sHomeSensorPortID,
									bEnableTimeout	:= TRUE,
									tDefaultTimeout	:= tGoHomeTimeout);
									
THIS^.piActiveSensor.MR_FirstCycleEx( 	sName			:= CONCAT(sName,':Active_Sensor'),
										sModuleType 	:= sActiveSensorModuleType,
										sPortID			:= sActiveSensorPortID,
										bEnableTimeout	:= TRUE,
										tDefaultTimeout	:= tGoActiveTimeout);
END_METHOD

METHOD MR_GoActive : BOOL
IF eCylinderState = CYLINDER_IDLE AND NOT piActiveSensor.In THEN
	bBusy := TRUE;
	bGoActive := TRUE;
	MR_GoActive := FALSE;
	eCylinderState := CYLINDER_GO_ACTIVE;
	eCylinderGoActiveState := CYLINDER_MOVE_START_TRACKING;
	fbMachineLogger.MR_AddLogs(CONCAT(sName,' : active position requested'));	
	
	
ELSIF eCylinderState = CYLINDER_GO_ACTIVE_DONE THEN
	bGoActive := FALSE;
	MR_GoActive := TRUE;
	fbMachineLogger.MR_AddLogs(CONCAT(sName,' : active position done'));		
	
END_IF
END_METHOD

METHOD MR_GoHome : BOOL
IF eCylinderState = CYLINDER_IDLE AND NOT piHomeSensor.In THEN
	bBusy := TRUE;
	bGoHome := TRUE;
	MR_GoHome := FALSE;
	eCylinderState := CYLINDER_GO_HOME;
	eCylinderGoHomeState := CYLINDER_MOVE_START_TRACKING;
	fbMachineLogger.MR_AddLogs(CONCAT(sName,' : home position requested'));	
	
ELSIF eCylinderState = CYLINDER_GO_HOME_DONE THEN
	bGoHome := FALSE;
	MR_GoHome := TRUE;
	fbMachineLogger.MR_AddLogs(CONCAT(sName,' : home position done'));	
	
END_IF
END_METHOD

METHOD MR_Init : BOOL
IF eCylinderState = CYLINDER_UNINITIALIZED THEN
	bBusy := TRUE;
	bInit := TRUE;
	MR_Init := FALSE;
	eCylinderState := CYLINDER_INITIALIZING;
	fbMachineLogger.MR_AddLogs(CONCAT(sName,' : initialization requested'));	
	
ELSIF eCylinderState = CYLINDER_IDLE THEN
	bInit := FALSE;
	MR_Init := TRUE;
	fbMachineLogger.MR_AddLogs(CONCAT(sName,' : initialization done'));	
	
END_IF
END_METHOD

METHOD MR_Release : BOOL
IF eCylinderState = CYLINDER_IDLE AND bPositionHold THEN
	bBusy := TRUE;
	bRelease := TRUE;
	MR_Release := FALSE;
	eCylinderState := CYLINDER_RELEASE;
	fbMachineLogger.MR_AddLogs(CONCAT(sName,' : release requested'));	
	
ELSIF eCylinderState = CYLINDER_RELEASE_DONE THEN	
	bRelease := FALSE;
	MR_Release := TRUE;
	fbMachineLogger.MR_AddLogs(CONCAT(sName,' : release done'));
	
END_IF
END_METHOD

METHOD MR_Reset : BOOL
IF eCylinderState >= CYLINDER_IDLE AND bError THEN
	bBusy := TRUE;
	bReset := TRUE;
	MR_Reset := FALSE;
	eCylinderState := CYLINDER_RESET;
	fbMachineLogger.MR_AddLogs(CONCAT(sName,' : reset requested'));	
	
ELSIF eCylinderState = CYLINDER_RESET_DONE THEN
	bReset := FALSE;
	MR_Reset := TRUE;
	fbMachineLogger.MR_AddLogs(CONCAT(sName,' : reset done'));		
	
END_IF
END_METHOD

METHOD PROTECTED  MS_Aborting
piHomeSensor.MR_Abort();
piActiveSensor.MR_Abort();

IF NOT piHomeSensor.Active AND NOT piActiveSensor.Active THEN
	//bBusy := FALSE;
	eCylinderState := CYLINDER_UNINITIALIZED;	
END_IF
END_METHOD

METHOD PROTECTED ABSTRACT MS_GoActive
END_METHOD

METHOD PROTECTED MS_GoActiveDone
IF NOT bGoActive THEN
	bBusy := FALSE;
	eCylinderState := CYLINDER_IDLE;
END_IF
END_METHOD

METHOD PROTECTED ABSTRACT MS_GoHome
END_METHOD

METHOD PROTECTED MS_GoHomeDone
IF NOT bGoHome THEN
	bBusy := FALSE;
	eCylinderState := CYLINDER_IDLE;
END_IF
END_METHOD

METHOD PROTECTED MS_Idle
;
END_METHOD

METHOD PROTECTED MS_Initializing
piHomeSensor.MR_Init();
piActiveSensor.MR_Init();

piHomeSensor.EnableTimeout := TRUE;
piActiveSensor.EnableTimeout := TRUE;

IF piHomeSensor.Active AND piActiveSensor.Active THEN
	eCylinderState := CYLINDER_READY_INITIALIZED;
END_IF
END_METHOD

METHOD PROTECTED MS_ReadyInitialized
VAR_INPUT
END_VAR
bBusy := FALSE;
eCylinderState := CYLINDER_IDLE;
END_METHOD

METHOD PROTECTED ABSTRACT MS_Release
END_METHOD

METHOD PROTECTED MS_ReleaseDone
IF NOT bRelease THEN
	bBusy := FALSE;
	eCylinderState := CYLINDER_IDLE;
END_IF
END_METHOD

METHOD PROTECTED MS_Reset
VAR_INPUT
END_VAR
bInit 		:= FALSE;
bGoActive 	:= FALSE;
bGoHome 	:= FALSE;
bRelease	:= FALSE;
bAbort		:= FALSE;

tonGoHomeDelay(IN := FALSE);
tonGoActiveDelay(IN := FALSE);
tonMeasurementTimer(IN:= FALSE);

piHomeSensor.MR_Reset();
piActiveSensor.MR_Reset();

IF NOT piHomeSensor.ErrorTimedout AND NOT piActiveSensor.ErrorTimedout THEN
	eCylinderState := CYLINDER_RESET_DONE;
END_IF
END_METHOD

METHOD PROTECTED MS_ResetDone
VAR_INPUT
END_VAR
IF NOT bReset THEN
	bBusy := FALSE;
	eCylinderState := CYLINDER_IDLE;
END_IF
END_METHOD

METHOD PROTECTED MS_Uninitialized
bError := FALSE;
bBusy := FALSE;

piHomeSensor.EnableForce := FALSE;
piActiveSensor.EnableForce := FALSE;

piHomeSensor.EnableTimeout := FALSE;
piActiveSensor.EnableTimeout := FALSE;

bInit 		:= FALSE;
bGoActive 	:= FALSE;
bGoHome 	:= FALSE;
bRelease	:= FALSE;
bReset		:= FALSE;
bAbort		:= FALSE;

tonGoHomeDelay(IN := FALSE);
tonGoActiveDelay(IN := FALSE);
tonMeasurementTimer(IN:= FALSE);
END_METHOD

PROPERTY Name : STRING
GET
Name := sName;
END_GET
SET
sName := Name;
END_SET
END_PROPERTY

PROPERTY PositionActive : REFERENCE TO BOOL
GET
PositionActive REF= bPositionActive;
END_GET
END_PROPERTY

PROPERTY PositionHold : REFERENCE TO BOOL
GET
PositionHold REF= bPositionHold;
END_GET
END_PROPERTY

PROPERTY PositionHome : REFERENCE TO BOOL
GET
PositionHome REF= bPositionHome;
END_GET
END_PROPERTY

PROPERTY ref_piActiveSensor : REFERENCE TO FB_DigitalInputExt
GET
ref_piActiveSensor REF= piActiveSensor;
END_GET
END_PROPERTY

PROPERTY ref_piHomeSensor : REFERENCE TO FB_DigitalInputExt
GET
ref_piHomeSensor REF= piHomeSensor;
END_GET
END_PROPERTY

PROPERTY Simulation : BOOL
GET
Simulation := bSimulation;
END_GET
SET
bSimulation := Simulation;
END_SET
END_PROPERTY

PROPERTY State : REFERENCE TO E_CylinderState
GET
State REF= eCylinderState;
END_GET
END_PROPERTY

METHOD PROTECTED StateMachine
CASE eCylinderState OF
	CYLINDER_UNINITIALIZED:
		MS_Uninitialized();
		
	CYLINDER_INITIALIZING:
		MS_Initializing();
	
	CYLINDER_READY_INITIALIZED:
		MS_ReadyInitialized();
		
	CYLINDER_IDLE:
		MS_Idle();
		
	CYLINDER_GO_HOME:
		MS_GoHome();
		
	CYLINDER_GO_HOME_DONE:
		MS_GoHomeDone();
		
	CYLINDER_GO_ACTIVE:
		MS_GoActive();
		
	CYLINDER_GO_ACTIVE_DONE:
		MS_GoActiveDone();
		
	CYLINDER_RELEASE:
		MS_Release();
		
	CYLINDER_RELEASE_DONE:
		MS_ReleaseDone();
		
	CYLINDER_RESET:
		MS_Reset();
		
	CYLINDER_RESET_DONE:
		MS_ResetDone();
		
	CYLINDER_ABORTING:
		MS_Aborting();
		
END_CASE
END_METHOD

END_FUNCTION_BLOCK

// ---- POUs/Libs/Digital Devices/Digital Input/FB_DigitalInputExt.TcPOU
(* 
| :Description: This function block represents basic digital input and can be used for creating an instance of signle digital input device like buttons, switches, sensors.
| To get the current status of digital input use "Value" property. To simulate state of the input by software set "Enable Force" parameter and change value via "MR_ResetForceValue" and "MR_SetForceValue" methods.
*)
FUNCTION_BLOCK FB_DigitalInputExt EXTENDS FB_DigitalInput
VAR
	(* Internal commands *)
	bInit 				: BOOL;		(*  *)
	bAbort				: BOOL;		(*  *)
	bReset				: BOOL;		(*  *)
	bTimeoutTracking	: BOOL;		(* Watchdog timer control bit *)
	
	(* Internal status *)
	bActive				: BOOL;		(*  *)
	bErrorTimedout		: BOOL;		(* Timeout coccured while waiting for signal *)
	eDigitalInputState	: E_DigitalInputExState;
	
	(*Internal parameters*)
	tTimeout			: TIME;		(* Input timeout *)
	bEnableTimeout		: BOOL;		(* Enable using timeout *)
	
	(* Function blocks *)
	bStartWatchdog		: BOOL;
	tonWatchdog			: TON;		(* Input timeout watchdog *)
	
END_VAR
(*
Version history:

+-------------+------------+----------------+----------+------------------------------------------+
|Date         | Version    | created under  | Author   | Remark                                   |
+=============+============+================+==========+==========================================+
|2022-03      | 1.0.0.0    | V3.1.4024.22   | ADBO     | Function block created                   |
+-------------+------------+----------------+----------+------------------------------------------+

*)

bActive := eDigitalInputState >= DIGITAL_INPUT_EX_IDLE; //OR eDigitalInputState = DIGITAL_INPUT_EX_ABORTING;

StateMachine();

tonWatchdog( IN := bStartWatchdog, PT := tTimeout);

PROPERTY Active : REFERENCE TO BOOL
GET
Active REF= bActive;
END_GET
END_PROPERTY

PROPERTY CurrentTimeout : REFERENCE TO TIME
GET
CurrentTimeout REF= tonWatchdog.ET;
END_GET
END_PROPERTY

PROPERTY EnableTimeout : BOOL
GET
EnableTimeout := bEnableTimeout;
END_GET
SET
bEnableTimeout := EnableTimeout;
END_SET
END_PROPERTY

PROPERTY ErrorTimedout : REFERENCE TO BOOL
GET
ErrorTimedout REF= bErrorTimedout;
END_GET
END_PROPERTY

METHOD MR_Abort : BOOL
VAR_INPUT
END_VAR
IF eDigitalInputState > DIGITAL_INPUT_EX_UNINITIALIZED THEN
	bAbort := TRUE;
	MR_Abort := FALSE;
	eDigitalInputState := DIGITAL_INPUT_EX_ABORTING;
	fbMachineLogger.MR_AddLogs(CONCAT(sName,' : abort requested'));	
	
ELSIF eDigitalInputState = DIGITAL_INPUT_EX_UNINITIALIZED THEN
	bAbort := FALSE;
	MR_Abort := TRUE;
	fbMachineLogger.MR_AddLogs(CONCAT(sName,' : abort done'));	
	
END_IF
END_METHOD

METHOD MR_FirstCycleEx : BOOL
VAR_INPUT
	sName			: STRING;
	sModuleType		: STRING;
	sPortID			: STRING;
	bEnableTimeout	: BOOL;
	tDefaultTimeout : TIME;
END_VAR
THIS^.sName := sName;
THIS^.ModuleType := sModuleType;
THIS^.PortID := sPortID;
THIS^.bEnableTimeout := bEnableTimeout;
THIS^.tTimeout := tDefaultTimeout;
END_METHOD

METHOD MR_Init : BOOL
VAR_INPUT
END_VAR
IF eDigitalInputState = DIGITAL_INPUT_EX_UNINITIALIZED THEN
	bInit := TRUE;
	MR_Init := FALSE;
	eDigitalInputState := DIGITAL_INPUT_EX_INITIALIZING;
	fbMachineLogger.MR_AddLogs(CONCAT(sName,' : initialization requested'));		
	
ELSIF eDigitalInputState = DIGITAL_INPUT_EX_IDLE AND bInit THEN
	bInit := FALSE;
	MR_Init := TRUE;
	fbMachineLogger.MR_AddLogs(CONCAT(sName,' : initialization done'));	

END_IF
END_METHOD

METHOD MR_Reset : BOOL
VAR_INPUT
END_VAR
IF eDigitalInputState = DIGITAL_INPUT_EX_IDLE THEN
	bReset := TRUE;
	MR_Reset := FALSE;
	eDigitalInputState := DIGITAL_INPUT_EX_RESET;
	fbMachineLogger.MR_AddLogs(CONCAT(sName,' : reset requested'));	
	
ELSIF eDigitalInputState = DIGITAL_INPUT_EX_RESET_DONE THEN
	bReset := FALSE;
	MR_Reset := TRUE;
	fbMachineLogger.MR_AddLogs(CONCAT(sName,' : reset done'));	
	
END_IF
END_METHOD

METHOD MR_StartTracking
VAR_INPUT
END_VAR
IF eDigitalInputState = DIGITAL_INPUT_EX_IDLE AND bEnableTimeout AND NOT bErrorTimedout THEN
	bTimeoutTracking := TRUE;
	eDigitalInputState := DIGITAL_INPUT_EX_TIMEOUT_TRACKING;
	fbMachineLogger.MR_AddLogs(CONCAT(sName,' : start tracking requested'));	
	
END_IF
END_METHOD

METHOD PROTECTED MS_Abort
VAR_INPUT
END_VAR
eDigitalInputState := DIGITAL_INPUT_EX_UNINITIALIZED;
END_METHOD

METHOD PROTECTED MS_Idle
VAR_INPUT
END_VAR
;
END_METHOD

METHOD PROTECTED MS_Initializing
VAR_INPUT
END_VAR
(* To-Do add alarm declaration *)

eDigitalInputState := DIGITAL_INPUT_EX_READY_INITIALIZED;
END_METHOD

METHOD PROTECTED MS_ReadyInitialized
VAR_INPUT
END_VAR
eDigitalInputState := DIGITAL_INPUT_EX_IDLE;
END_METHOD

METHOD PROTECTED MS_Reset
VAR_INPUT
END_VAR
bErrorTimedout := FALSE;
eDigitalInputState := DIGITAL_INPUT_EX_RESET_DONE;
END_METHOD

METHOD PROTECTED MS_ResetDone
VAR_INPUT
END_VAR
IF NOT bReset THEN
	eDigitalInputState := DIGITAL_INPUT_EX_IDLE;
END_IF
END_METHOD

METHOD PROTECTED MS_TimeoutTracking
VAR_INPUT
END_VAR
IF tonWatchdog.Q THEN
	(* To-Do raise alarm *)
	bErrorTimedout := TRUE;
	bStartWatchdog := FALSE;
	eDigitalInputState := DIGITAL_INPUT_EX_TIMEOUT_TRACKING_DONE;
	
ELSE
	bStartWatchdog := TRUE;
	
	IF bRisingTrigger OR bFallingTrigger THEN
		bStartWatchdog := FALSE;
		eDigitalInputState := DIGITAL_INPUT_EX_TIMEOUT_TRACKING_DONE;
	
	END_IF
END_IF
END_METHOD

METHOD PROTECTED MS_TimeoutTrackingDone
VAR_INPUT
END_VAR
bTimeoutTracking := FALSE;
eDigitalInputState := DIGITAL_INPUT_EX_IDLE;
END_METHOD

METHOD PROTECTED MS_Uninitialized
VAR_INPUT
END_VAR
bInit := FALSE;
bAbort := FALSE;
bReset := FALSE;
bTimeoutTracking := FALSE;

bRisingTrigger := FALSE;
bFallingTrigger := FALSE;
bErrorTimedout := FALSE;

tonWatchdog( IN := FALSE, PT := tTimeout);
END_METHOD

PROPERTY State : REFERENCE TO E_DigitalInputExState
GET
State REF= eDigitalInputState;
END_GET
END_PROPERTY

METHOD PROTECTED StateMachine
VAR_INPUT
END_VAR
CASE eDigitalInputState OF
	DIGITAL_INPUT_EX_UNINITIALIZED:
		MS_Uninitialized();
		
	DIGITAL_INPUT_EX_INITIALIZING:
		MS_Initializing();
		
	DIGITAL_INPUT_EX_READY_INITIALIZED:
		MS_ReadyInitialized();
		
	DIGITAL_INPUT_EX_IDLE:
		MS_Idle();
		
	DIGITAL_INPUT_EX_TIMEOUT_TRACKING:
		MS_TimeoutTracking();	
	
	DIGITAL_INPUT_EX_TIMEOUT_TRACKING_DONE:
		MS_TimeoutTrackingDone();	
	
	DIGITAL_INPUT_EX_RESET:
		MS_Reset();

	DIGITAL_INPUT_EX_RESET_DONE:
		MS_ResetDone();
	
	DIGITAL_INPUT_EX_ABORTING:
		MS_Abort();
	
END_CASE
END_METHOD

PROPERTY Timeout : TIME
GET
Timeout := tTimeout;
END_GET
SET
tTimeout := Timeout;
END_SET
END_PROPERTY

END_FUNCTION_BLOCK

// ---- POUs/Libs/Digital Devices/Digital Output/FB_DigitalOutput.TcPOU
(* 
| :Description: This function block represents basic digital output and can be used for creating an instance of signle digital output device. 
| To control the output state use property "Value" 
*)
FUNCTION_BLOCK FB_DigitalOutput EXTENDS FB_DigitalDevice IMPLEMENTS  I_DigitalOutput
VAR
	bOut AT %Q*: BOOL; (* Current value of output*)
END_VAR
(*
Version history:

+-------------+------------+----------------+----------+------------------------------------------+
|Date         | Version    | created under  | Author   | Remark                                   |
+=============+============+================+==========+==========================================+
|2021-11      | 1.0.0.0    | V3.1.4024.22   | ADBO     | Function block created                   |
+-------------+------------+----------------+----------+------------------------------------------+
|2022-02      | 1.1.0.0    | V3.1.4024.22   | ADBO     | Changed to child of FB_DigitalDevice     |
+-------------+------------+----------------+----------+------------------------------------------+

*)

PROPERTY Out : BOOL
GET
Out := bOut;
END_GET
SET
bOut := Out;
END_SET
END_PROPERTY

END_FUNCTION_BLOCK

// ---- POUs/Libs/Cylinder/Double Coil Cylinder/FB_DoubleCoilCylinder2.TcPOU
FUNCTION_BLOCK FB_DoubleCoilCylinder2 EXTENDS FB_SingleCoilCylinder
VAR_INPUT
END_VAR
VAR_OUTPUT
END_VAR
VAR
	(* Coils *)
	poHomeValve	: FB_DigitalOutput;	(* Home position valve function block *)
END_VAR

IF bFirstCycle THEN
	poActiveValve.MR_FirstCycle( sName := CONCAT(sName,':Home_Valve'),sModuleType := ref_poHomeValve.ModuleType, sPortID := ref_poHomeValve.PortID);	
END_IF

SUPER^();

bPositionHold := poActiveValve.Out OR poHomeValve.Out;

poHomeValve();

METHOD MR_GoActive : BOOL
IF eCylinderState = CYLINDER_IDLE AND NOT poActiveValve.Out THEN
	bBusy := TRUE;
	bGoActive := TRUE;
	MR_GoActive := FALSE;
	eCylinderState := CYLINDER_GO_ACTIVE;
	eCylinderGoActiveState := CYLINDER_MOVE_START_TRACKING;
	fbMachineLogger.MR_AddLogs(CONCAT(sName,' : active position requested'));	
	
	
ELSIF eCylinderState = CYLINDER_GO_ACTIVE_DONE THEN
	bGoActive := FALSE;
	MR_GoActive := TRUE;
	fbMachineLogger.MR_AddLogs(CONCAT(sName,' : active position done'));		
	
END_IF
END_METHOD

METHOD MR_GoHome : BOOL
IF eCylinderState = CYLINDER_IDLE AND NOT poHomeValve.Out THEN
	bBusy := TRUE;
	bGoHome := TRUE;
	MR_GoHome := FALSE;
	eCylinderState := CYLINDER_GO_HOME;
	eCylinderGoHomeState := CYLINDER_MOVE_START_TRACKING;
	fbMachineLogger.MR_AddLogs(CONCAT(sName,' : home position requested'));	
	
ELSIF eCylinderState = CYLINDER_GO_HOME_DONE THEN
	bGoHome := FALSE;
	MR_GoHome := TRUE;
	fbMachineLogger.MR_AddLogs(CONCAT(sName,' : home position done'));	
	
END_IF
END_METHOD

METHOD PROTECTED MS_GoActive
VAR_INPUT
END_VAR
poHomeValve.Out := FALSE;
SUPER^.MS_GoActive();
END_METHOD

METHOD PROTECTED MS_GoHome
VAR_INPUT
END_VAR
poHomeValve.Out := TRUE;
SUPER^.MS_GoHome();
END_METHOD

METHOD PROTECTED MS_Release
VAR_INPUT
END_VAR
poHomeValve.Out := FALSE;
SUPER^.MS_Release();
END_METHOD

METHOD PROTECTED MS_Reset
VAR_INPUT
END_VAR
poHomeValve.Out := FALSE;

SUPER^.MS_Reset();
END_METHOD

METHOD PROTECTED MS_Uninitialized
poHomeValve.Out := FALSE;
SUPER^.MS_Uninitialized();
END_METHOD

PROPERTY ref_poHomeValve : REFERENCE TO FB_DigitalOutput
GET
ref_poHomeValve REF= poHomeValve;
END_GET
END_PROPERTY

END_FUNCTION_BLOCK

// ---- POUs/Libs/Cylinder/Single Coil Cylinder/FB_SingleCoilCylinder2.TcPOU
FUNCTION_BLOCK FB_SingleCoilCylinder2 EXTENDS FB_UniversalCylinder
VAR_INPUT
	
END_VAR
VAR_OUTPUT
END_VAR
VAR
	(* Coils *)
	poActiveValve	: FB_DigitalOutput;	(* Active position valve function block *)
END_VAR

IF bFirstCycle THEN
	poActiveValve.MR_FirstCycle( sName := CONCAT(sName,':Active_Valve'),sModuleType := ref_poActiveValve.ModuleType, sPortID:= ref_poActiveValve.PortID);
END_IF

SUPER^();

bPositionHold := poActiveValve.Out;

poActiveValve();

METHOD PROTECTED M_SimulationLogic
VAR_INPUT
END_VAR
IF poActiveValve.Out THEN
	piActiveSensor.MR_SetForceValue();
	piHomeSensor.MR_ResetForceValue();
	
ELSIF NOT poActiveValve.Out THEN
	piActiveSensor.MR_ResetForceValue();
	piHomeSensor.MR_SetForceValue();
	
END_IF
END_METHOD

METHOD MR_GoActive : BOOL
IF eCylinderState = CYLINDER_IDLE AND NOT poActiveValve.Out THEN
	bBusy := TRUE;
	bGoActive := TRUE;
	MR_GoActive := FALSE;
	eCylinderState := CYLINDER_GO_ACTIVE;
	eCylinderGoActiveState := CYLINDER_MOVE_START_TRACKING;
	fbMachineLogger.MR_AddLogs(CONCAT(sName,' : active position requested'));	
	
	
ELSIF eCylinderState = CYLINDER_GO_ACTIVE_DONE THEN
	bGoActive := FALSE;
	MR_GoActive := TRUE;
	fbMachineLogger.MR_AddLogs(CONCAT(sName,' : active position done'));		
	
END_IF
END_METHOD

METHOD MR_GoHome : BOOL
IF eCylinderState = CYLINDER_IDLE AND poActiveValve.Out THEN
	bBusy := TRUE;
	bGoHome := TRUE;
	MR_GoHome := FALSE;
	eCylinderState := CYLINDER_GO_HOME;
	eCylinderGoHomeState := CYLINDER_MOVE_START_TRACKING;
	fbMachineLogger.MR_AddLogs(CONCAT(sName,' : home position requested'));	
	
ELSIF eCylinderState = CYLINDER_GO_HOME_DONE THEN
	bGoHome := FALSE;
	MR_GoHome := TRUE;
	fbMachineLogger.MR_AddLogs(CONCAT(sName,' : home position done'));	
	
END_IF
END_METHOD

METHOD PROTECTED MS_GoActive
VAR_INPUT
END_VAR
poActiveValve.Out := TRUE;

CASE eCylinderGoActiveState OF
	CYLINDER_MOVE_START_TRACKING:
		piActiveSensor.MR_StartTracking();
		
		IF piActiveSensor.In THEN
			IF TIME_TO_INT(tDelay) = 0 THEN
				eCylinderGoActiveState := CYLINDER_MOVE_DONE;
			ELSE
				eCylinderGoActiveState := CYLINDER_MOVE_DELAY;
			END_IF
		END_IF
		
	CYLINDER_MOVE_DELAY:
		tonGoActiveDelay( IN := TRUE, PT := tDelay);
		
		IF tonGoActiveDelay.Q THEN
			tonGoActiveDelay( IN := FALSE );
			eCylinderGoActiveState := CYLINDER_MOVE_DONE;
		END_IF
		
	CYLINDER_MOVE_DONE:
		eCylinderState := CYLINDER_GO_ACTIVE_DONE;
		
END_CASE
END_METHOD

METHOD PROTECTED MS_GoHome
VAR_INPUT
END_VAR
poActiveValve.Out := FALSE;

CASE eCylinderGoHomeState OF
	CYLINDER_MOVE_START_TRACKING:
		piHomeSensor.MR_StartTracking();
		
		IF piHomeSensor.In THEN
			IF TIME_TO_INT(tDelay) = 0 THEN
				eCylinderGoHomeState := CYLINDER_MOVE_DONE;
			ELSE
				eCylinderGoHomeState := CYLINDER_MOVE_DELAY;
			END_IF
		END_IF
		
	CYLINDER_MOVE_DELAY:
		tonGoHomeDelay( IN := TRUE, PT := tDelay);
		
		IF tonGoHomeDelay.Q THEN
			tonGoHomeDelay( IN := FALSE);
			eCylinderGoHomeState := CYLINDER_MOVE_DONE;
		END_IF
		
	CYLINDER_MOVE_DONE:
		eCylinderState := CYLINDER_GO_HOME_DONE;
	
END_CASE
END_METHOD

METHOD PROTECTED MS_Release
VAR_INPUT
END_VAR
poActiveValve.Out := FALSE;
eCylinderState := CYLINDER_RELEASE_DONE;
END_METHOD

METHOD PROTECTED MS_Reset
VAR_INPUT
END_VAR
poActiveValve.Out := FALSE;

SUPER^.MS_Reset();
END_METHOD

METHOD PROTECTED MS_Uninitialized
poActiveValve.Out := FALSE;
SUPER^.MS_Uninitialized();
END_METHOD

PROPERTY ref_poActiveValve : REFERENCE TO FB_DigitalOutput
GET
ref_poActiveValve REF= poActiveValve;
END_GET
END_PROPERTY

END_FUNCTION_BLOCK

// ---- POUs/Libs/Digital Devices/Lamp Indicator/FB_Lamp.TcPOU
(* 
:Description: 
*)
FUNCTION_BLOCK FB_Lamp EXTENDS FB_DigitalDevice IMPLEMENTS I_Lamp
VAR
	bFirstCycle : BOOL := TRUE;
	
	poLamp				: FB_DigitalOutput;		(*  *)
	eLampState			: E_LampState;			(*  *)
	tonBlinkingTimer	: TON;					(*  *)
	tBlinkTime			: TIME;					(*  *)
	In: INT;
END_VAR
(*
Version history:

+-------------+------------+----------------+----------+------------------------------------------+
|Date         | Version    | created under  | Author   | Remark                                   |
+=============+============+================+==========+==========================================+
|2021-11      | 1.0.0.0    | V3.1.4024.22   | ADBO     | Function block created                   |
+-------------+------------+----------------+----------+------------------------------------------+

*)

IF bFirstCycle THEN
	bFirstCycle := FALSE;
	poLamp.MR_FirstCycle(CONCAT('Digital output of: ',sName),sModuleType,sPortID);
END_IF

(*  *)
tonBlinkingTimer(	IN := (eLampState = LAMP_BLINKING_ON OR 
					eLampState = LAMP_BLINKING_OFF) AND NOT tonBlinkingTimer.Q,
					PT := tBlinkTime);

(*  *)
StateMachine();

(* *)
poLamp.Out := (eLampState = LAMP_ON OR eLampState = LAMP_BLINKING_ON);

METHOD MR_LampBlink : BOOL
VAR_INPUT
	tBlinkTime : TIME;
END_VAR
THIS^.tBlinkTime := tBlinkTime;

IF eLampState = LAMP_OFF THEN
	eLampState := LAMP_BLINKING_ON;
	
ELSIF eLampState = LAMP_ON THEN
	eLampState := LAMP_BLINKING_OFF;
	
END_IF

MR_LampBlink := TRUE;
END_METHOD

METHOD MR_LampOff : BOOL
eLampState := LAMP_OFF;
MR_LampOff := TRUE;
END_METHOD

METHOD MR_LampOn : BOOL
eLampState := LAMP_ON;
MR_LampOn := TRUE;
END_METHOD

METHOD PROTECTED MS_LampBlinkingOff
VAR_INPUT
END_VAR
IF tonBlinkingTimer.Q THEN
	eLampState := LAMP_BLINKING_ON;
END_IF
END_METHOD

METHOD PROTECTED MS_LampBlinkingOn
VAR_INPUT
END_VAR
IF tonBlinkingTimer.Q THEN
	eLampState := LAMP_BLINKING_OFF;
END_IF
END_METHOD

METHOD PROTECTED MS_LampOff
VAR_INPUT
END_VAR
;
END_METHOD

METHOD PROTECTED MS_LampOn
VAR_INPUT
END_VAR
;
END_METHOD

METHOD PROTECTED StateMachine
VAR_INPUT
END_VAR
(*  *)
CASE eLampState OF
	LAMP_OFF:
		MS_LampOff();
		
	LAMP_ON:
		MS_LampOn();
		
	LAMP_BLINKING_ON:
		MS_LampBlinkingOn();
		
	LAMP_BLINKING_OFF:
		MS_LampBlinkingOff();
	
END_CASE
END_METHOD

PROPERTY Status : REFERENCE TO E_LampState
GET
Status REF= eLampState;
END_GET
END_PROPERTY

END_FUNCTION_BLOCK

// ---- POUs/Libs/Fixtures/FB_UniversalFixture.TcPOU
(* 
:Description: This function block is base for all other measurement fixtures.
*)
FUNCTION_BLOCK ABSTRACT FB_UniversalFixture IMPLEMENTS  I_UniversalFixture
VAR CONSTANT
	sSAMPLE_ACCEPTED : STRING := 'ACCEPTED';					(* Sample accepted - compare keyword for TCP/IP message from measurement device *)
	sSAMPLE_REJECTED : STRING := 'REJECTED';					(* Sample rejected - compare keyword for TCP/IP message from measurement device *)
END_VAR
VAR
	bFirstCycle				: BOOL := TRUE;						(* First cycle bit *)
	sName 					: STRING; 							(* Fixture name for other utilities *)
	
	bActive 				: BOOL;								(* Fixture device is initialized and ready to wokr *)
	bBusy					: BOOL;								(* Fixture device is busy *)
	bError 					: BOOL;								(* Error occured while executing *)
	iErrorID 				: UDINT;							(* Error ID *)
	
	eSampleResult			: E_UniversalFixtureSampleResult;	(* Result of current measured product *)
	iSampleID				: UDINT;							(* Id of current measured product *)
	bSocketOpen				: BOOL;								(* Socket open flag *)
	
	sSendData				: STRING;							(* String message to send via TCP/IP to measurement device *)
	sRecivedData			: STRING;							(* String message to recive via TCP/IP from measurement device *)
	sLoggerMessage			: STRING;							(* String message for measurement txt logger *)
	stSendData				: ST_TcpBufferData;					(* Byte message to send via TCP/IP to measurement device *)
	stReciveData			: ST_TcpBufferData;					(* Byte message to recive via TCP/IP from measurement device *)
	fbTcpServer				: FB_TcpServer;						(* TCP/IP server instance *)
	fbTcpClient				: FB_TcpClient;						(* TCP/IP client instance *)
	bUseLogger				: BOOL;								(* Enables using of internal fixture file logger *)
	fbMeasurementLogger 	: FB_TXTDataExchanger;				(* Measurement TXT-File logger *)
	
	rtError					: R_TRIG; 							(* Rising edge trigger for function block error *)
	
	eFixtureState			: E_UniversalFixtureState;			(* Current state of measurement fixture device *)
	eFixtureStateInit		: E_UniversalFixtureStateInit;		(* Current state of measurement fixture device initialization *)
	eFixtureStateAbort		: E_UniversalFixtureStateAbort;		(* Current state of measurement fixture device aborting *)
	eFixtureStateReset		: E_UniversalFixtureStateReset;		(* Current state of measurement fixture device reseting *)
	eFixtureStateMeasure	: E_UniversalFixtureStateMeasure; 	(* Current measurement state if measurement has began *)
	eConnnectionType		: E_UniversalFixtureConnectionType;
	
	bClientConnection 		: BOOL; 							(* If true then fixture connect as a client, if false it behaves like a server *)
END_VAR

(* First cycle assignamnets *)
IF bFirstCycle THEN
	bFirstCycle := FALSE;
	
END_IF

(* Update status flags *)
bActive := eFixtureState >= UNIVERSAL_FIXTURE_READY;
bError := fbTcpServer.Error OR fbMeasurementLogger.Error;

(* Run server instance *)
IF eConnnectionType = UNIVERSAL_FIXTURE_SERVER_CONNECTION THEN
	fbTcpServer();
	
ELSIF eConnnectionType = UNIVERSAL_FIXTURE_CLIENT_CONNECTION THEN
	fbTcpClient();
	
END_IF 

(* Report errors that occur *)
rtError(CLK:=bError);

IF rtError.Q THEN 
	fbMachineLogger.MR_AddLogs(FUN_MergeStrings5(sName, ' : Error occured (error ID: ', UDINT_TO_STRING(iErrorID), ')', ''));
	
END_IF

(* Run internal measurement logger instance if it's enabled *)
IF bUseLogger THEN
	fbMeasurementLogger();
	
END_IF

(* Run main state machine *)
StateMachine();

PROPERTY Active : REFERENCE TO BOOL
GET
Active REF= bActive;
END_GET
END_PROPERTY

PROPERTY Busy : REFERENCE TO BOOL
GET
Busy REF= bBusy;
END_GET
END_PROPERTY

PROPERTY Error : REFERENCE TO BOOL
GET
Error REF= bError;
END_GET
END_PROPERTY

